# B&R Automation Studio project BaseProject
Automation Studio 4.9.2.46; technology packages: mapp 5.15.0, mappCockpit 5.15.0, mappMotion 5.15.1, mappView 5.15.1

## Configuration BuildConfig

CPU PC_any, AutomationRuntime C4.90, Build 6.3.0, Safety 0.0, Vc 

### Task classes (Cpu.sw)
```
Cyclic#8 (cycle 9600 us):
  TrakDiag <- Source.Diagnostic.TrakDiag.prg
DataObjects: McAcpSys
Binaries: McAcpDrv, udbdef, McAcpSim, mvLoader, arflatprv, McProfGen, TCLang, TCData, FWRules, mCoWebSc, arcoal, arsvcreg, McMechSys, OpcUaSrv, sysconf, Settings, FileCfg, asfw, MainAlrCfg, MachCfg, Role, ashwac, TraceConfi, iomap, AlarmHist, SectorCfg, arconfig, AsmCfg, TC, ashwd, User, ShuttleCfg, AsmFeatCfg, CoreCfg, LoggerCFG, Main, AuditCfg, Config, em2_sm2, em2_sm1, Trak
Libraries: CoTrace, AsZip, FileIO, runtime, McBase, MpAlarmX, MpBase, astime, MpFile, MpRecipe, sys_lib, McAxis, McAcpTrak, MpAxis, McAcpAx, TrBase, MpPackML, MpCom, MpServer, MpRobotics, McAxGroup, McPathGen, McProgInt, snprintf, brdkSTR, TrkPaper, ArEventLog, AsHttp, AsIODiag, AsBrStr, standard, MpAudit, McAcpPar, AdvIecChk, asstring, TrkDiag, powerlnk, asieccon, asepl, asusb, dataobj, arssl, aruser, asarprof, asmem, brsystem, asarlog, asio
```

### Hardware
```
5PC910.SX02-00 : 5PC910.SX02-00 v2.0.1.0
  Connector IF1:
    AssignedOperatingSystem = ARemb
  Connector IF3:
    AssignedOperatingSystem = ARemb
    ActivateDevice = 1
    HostName = atldemo2019
    Mode = DHCP Server
  Connector IF4:
    AssignedOperatingSystem = ARemb
    ActivateDevice = 1
    HostName = atldemo2019
    Mode = Manual
    InternetAddress = 10.1.13.45
    SubnetMask = 255.255.255.0
  Connector IF5:
    AssignedOperatingSystem = ARemb
  Connector IF6:
    AssignedOperatingSystem = ARemb
  Connector IF7:
    AssignedOperatingSystem = ARemb
  Connector IF8:
    AssignedOperatingSystem = ARemb
  Connector IF9:
    AssignedOperatingSystem = ARemb
PC : 5PC900.TS17-00 v2.1.0.0  [SY -> 5PC910.SX02-00.SY1]
  ConfigurationID = BaseProject_TestConfig
  ConfigVersion = 1.2.0
  UserPartitionSize = 1024
  Simulation = 1
  VolatileGlobalPvSize = 2000000
  SystemTick = 400
  IdleTaskClass = 3
  TaskClassIdleTime = 2400
  XLinkUseDefault = 0
  XLinkDuration = 800
  Cyclic1Duration = 800
  Cyclic1Tolerance = 0
  Cyclic1Stack = 256000
  Cyclic1Output = 1
  Cyclic2Duration = 16000
  Cyclic2Tolerance = 32000
  Cyclic2Stack = 32000
  Cyclic3Duration = 49600
  Cyclic3Tolerance = 49600
  Cyclic8Duration = 9600
  FileDevice1
  FileDeviceName1 = SvgData
  FileDevicePath1 =  ../../../../Logical/Scene/
  FileDevice2
  FileDeviceName2 = User
  FileDevicePath2 = F:\
  FileDevice3
  FileDeviceName3 = Config
  FileDevicePath3 = F:\Config\
  FileDevice4
  FileDeviceName4 = SegTraceSim
  FileDevicePath4 = ../../../../Logical/UserData/SegTrace
  FileDevice5
  FileDeviceName5 = SegTrace
  FileDevicePath5 = F:/SegTrace
  FtpUser1
  FtpUsername1 = FTP
  FtpUserPassword1 = T9zhCndb3U+RGv/CzHF4XnaM0UkBa3EbnmIr44HqX4c=  // ftpaccess
  FtpUserSalt1 = Ims2GQYk
  FTPAccessRight1 = 0
  ActivateOpcUa = 1
  OpcUaInformationModels_PV_Version = 1
```

### LoggerCFG.mappmotioncfg - PC/mappMotion/LoggerCFG.mappmotioncfg
```
Element MappMotionConfiguration (Type=mappmotioncfg)
  Logger:
    SelectiveLogging = Used
      AdministrativeCommands = Suppressed
      MovementCommands = Suppressed
      InformationalCommands = Suppressed
```

### AsmCfg.assembly - PC/mappMotion/TrakConfig/AsmCfg.assembly
```
Element gSampleTrak (Type=assembly)
  Tracks:
    TrackSeparation = 0.030
    Track[1]:
      Segments:
        SegmentRef[1] = ::gSeg_A_1
        SegmentRef[2] = ::gSeg_A_2
        SegmentRef[3] = ::gSeg_A_3
        SegmentRef[4] = ::gSeg_A_4
        SegmentRef[5] = ::gSeg_A_5
        SegmentRef[6] = ::gSeg_A_6
        SegmentRef[7] = ::gSeg_A_7
        SegmentRef[8] = ::gSeg_A_8
        SegmentRef[9] = ::gSeg_A_9
        SegmentRef[10] = ::gSeg_A_10
        SegmentRef[11] = ::gSeg_A_11
        SegmentRef[12] = ::gSeg_A_12
      Position = Absolute
        SegmentRef = ::gSeg_A_1
        SegmentCountDirection = RightToLeft
        Translation:
          X = 0.0
          Y = 0.0
          Z = 0.0
        Orientation:
          Angle1 = 0.0
          Angle2 = 0.0
          Angle3 = 0.0
    Track[2]:
      Segments:
        SegmentRef[1] = ::gSeg_B_1
        SegmentRef[2] = ::gSeg_B_2
        SegmentRef[3] = ::gSeg_B_3
        SegmentRef[4] = ::gSeg_B_4
        SegmentRef[5] = ::gSeg_B_5
        SegmentRef[6] = ::gSeg_B_6
        SegmentRef[7] = ::gSeg_B_7
        SegmentRef[8] = ::gSeg_B_8
        SegmentRef[9] = ::gSeg_B_9
        SegmentRef[10] = ::gSeg_B_10
        SegmentRef[11] = ::gSeg_B_11
      Position = RelativeToOne
        TrackSegmentPosition:
          SegmentRef = ::gSeg_B_1
        Base:
          SegmentRef = ::gSeg_A_7
  CommonSegmentSettings:
    SegmentSimulationOnPLC = Off
    ElongationCompensation = Inactive
    StopReaction = InductionHalt
    SpeedFilter = Lowpass
      FilterTime = 0.0008
    ControllerParameters:
      DefaultParameter:
        Controller:
          Position:
            ProportionalGain = 150
          Speed:
            ProportionalGain = 80
            IntegrationTime = 0.0
          FeedForward:
            TotalMass = 0.7
            ForcePositive = 1.5
            ForceNegative = 1.5
            SpeedForceFactor = 1.4
            ForceLoad = 0.0
        MovementErrorLimits:
          PositionError = 20
          VelocityError = 2000
      AdditionalParameterSets = NotUsed
    ScopeOfErrorReaction = Assembly
    ShuttleIdentificationTime = 0
  Shuttles:
    MaxShuttleCount = 20
    DistanceReserve:
      Collision = 0.002
      ErrorStop = 0.006
    ShuttleStereotypes:
      ShuttleStRef[1] = gSampleShuttle
    MagnetPlateConfigurations:
      ShuttleType[1] = 8F1SA.100.xxxxxx-x
    CollisionAvoidance:
      Strategy = Constant
      MaximumModelDimensions:
        Length:
          ExtentToFront = 0.025
          ExtentToBack = 0.025
        Width:
          Width = 0.040
  AssemblyFeatures:
    AssemblyFeatureRef[1] = SampleTrak_AutoAttach
    AssemblyFeatureRef[2] = SampleTrak_LocalLimits
    AssemblyFeatureRef[3] = SampleTrak_SimShuttle
  Visualization:
    MonitoringPv = ::gSampleTrakMon
    ProcessingTaskClass = 1
```

### AsmFeatCfg.assemblyfeature - PC/mappMotion/TrakConfig/AsmFeatCfg.assemblyfeature
```
Element SampleTrak_AutoAttach (Type=assemblyfeature)
  Type = ShtSectorAutoAttach
    Priority[1]:
      SectorRef = gSampleTrak_SectorTrakA
      Orientation = KeepSegment
Element SampleTrak_LocalLimits (Type=assemblyfeature)
  Type = LocalLimits
    LocalLimit[1]:
      Location:
        SectorRef = gSampleTrak_SectorTrakA
      MotionLimits:
        Velocity = Basic
          Velocity = 3
        Acceleration = Basic
          Acceleration = 10
Element SampleTrak_SimShuttle (Type=assemblyfeature)
  Type = InitShuttleSim
    InitShuttleSim[1]:
      SectorRef = gSampleTrak_SectorTrakA
      Orientation = Positive
      ShuttleDefinition = ShuttleSetDefinition
        StartPosition = 0.0
        NumberOfShuttles = 10
        DistnaceBetweenShuttles = 100
```

### SectorCfg.sector - PC/mappMotion/TrakConfig/SectorCfg.sector
```
Element gSampleTrak_SectorTrakB (Type=sector)
  Type = Composed
    StartSegment:
      SegmentRef = ::gSeg_B_1
    IntermediateSegments:
      SegmentRef[1] = ::gSeg_B_2
      SegmentRef[2] = ::gSeg_B_3
      SegmentRef[3] = ::gSeg_B_4
      SegmentRef[4] = ::gSeg_B_5
      SegmentRef[5] = ::gSeg_B_6
      SegmentRef[6] = ::gSeg_B_7
      SegmentRef[7] = ::gSeg_B_8
      SegmentRef[8] = ::gSeg_B_9
      SegmentRef[9] = ::gSeg_B_10
    EndSegment:
      SegmentRef = ::gSeg_B_11
      PositionRelativeTo = FromEnd
Element gSampleTrak_SectorTrakAll (Type=sector)
  Type = Composed
    StartSegment:
      SegmentRef = ::gSeg_B_4
    IntermediateSegments:
      SegmentRef[1] = ::gSeg_B_5
      SegmentRef[2] = ::gSeg_B_6
      SegmentRef[3] = ::gSeg_B_7
      SegmentRef[4] = ::gSeg_B_8
      SegmentRef[5] = ::gSeg_B_9
      SegmentRef[6] = ::gSeg_B_10
      SegmentRef[7] = ::gSeg_B_11
      SegmentRef[8] = ::gSeg_A_7
      SegmentRef[9] = ::gSeg_A_6
      SegmentRef[10] = ::gSeg_A_5
      SegmentRef[11] = ::gSeg_A_4
      SegmentRef[12] = ::gSeg_A_3
      SegmentRef[13] = ::gSeg_A_2
      SegmentRef[14] = ::gSeg_A_1
      SegmentRef[15] = ::gSeg_A_12
      SegmentRef[16] = ::gSeg_A_11
      SegmentRef[17] = ::gSeg_A_10
      SegmentRef[18] = ::gSeg_A_9
      SegmentRef[19] = ::gSeg_A_8
      SegmentRef[20] = ::gSeg_A_7
      SegmentRef[21] = ::gSeg_B_1
      SegmentRef[22] = ::gSeg_B_2
      SegmentRef[23] = ::gSeg_B_3
    EndSegment:
      SegmentRef = ::gSeg_B_4
Element gSampleTrak_SectorTrakA (Type=sector)
  Type = Composed
    StartSegment:
      SegmentRef = ::gSeg_A_1
    IntermediateSegments:
      SegmentRef[1] = ::gSeg_A_2
      SegmentRef[2] = ::gSeg_A_3
      SegmentRef[3] = ::gSeg_A_4
      SegmentRef[4] = ::gSeg_A_5
      SegmentRef[5] = ::gSeg_A_6
      SegmentRef[6] = ::gSeg_A_7
      SegmentRef[7] = ::gSeg_A_8
      SegmentRef[8] = ::gSeg_A_9
      SegmentRef[9] = ::gSeg_A_10
      SegmentRef[10] = ::gSeg_A_11
    EndSegment:
      SegmentRef = ::gSeg_A_12
      PositionRelativeTo = FromEnd
```

### AlarmHist.mpalarmxhistory - PC/mappServices/Alarm/AlarmHist.mpalarmxhistory
```
Element gAlarmXHistory (Type=mpalarmxhistory)
```

### FileCfg.mpfilemanager - PC/mappServices/MachineConfig/FileCfg.mpfilemanager
```
Element FileManagement (Type=mpfilemanager)
  FileManager:
    USB = 1
```

### CoreCFG.mppackmlcore - PC/mappServices/Operation/CoreCFG.mppackmlcore
```
Element gPackMLCore (Type=mppackmlcore)
  Operation:
    Mode = 0
  Modes:
    Mode[1]:
      ModeID = 1
      Name = Production
  Unit:
    StartupActiveMode = 1
  UnitModes:
    Mode[1]:
      ModeID = 1
  Alarms = MpAlarmX
```

## Configuration TestConfig

CPU PC_any, AutomationRuntime C4.90, Build 6.3.0, Safety 0.0, Vc 

### Task classes (Cpu.sw)
```
Cyclic#1 (cycle 800 us, tolerance 0 us):
  GlobalSetu <- Source.GlobalSetup.prg
  TSM <- Source.TSM.prg
Cyclic#2 (cycle 1600 us, tolerance 0 us):
  TSMMain <- Source.TSMMain.prg
Cyclic#3:
  TSMAlarm <- Source.TSMAlarm.prg
DataObjects: McAcpSys
Binaries: McAcpDrv, udbdef, McAcpSim, mvLoader, arflatprv, McProfGen, TCLang, TCData, FWRules, mCoWebSc, arcoal, arsvcreg, McMechSys, sysconf, Settings, FileCfg, asfw, MainAlrCfg, MachCfg, Role, ashwac, TraceConfi, iomap, AlarmHist, SectorCfg, arconfig, AsmCfg, TC, ashwd, User, ShuttleCfg, AsmFeatCfg, CoreCfg, LoggerCFG, Main, AuditCfg, Config, em2_sm2, em2_sm1, Trak
Libraries: CoTrace, AsZip, FileIO, runtime, McBase, MpAlarmX, MpBase, astime, MpFile, MpRecipe, sys_lib, McAxis, McAcpTrak, MpAxis, McAcpAx, TrBase, MpPackML, MpCom, MpServer, MpRobotics, McAxGroup, McPathGen, McProgInt, snprintf, brdkSTR, TrkPaper, ArEventLog, AsHttp, AsIODiag, AsBrStr, standard, MpAudit, McAcpPar, AdvIecChk, asstring, TrkDiag, powerlnk, asieccon, asepl, asusb, dataobj, arssl, aruser, asarprof, asmem, brsystem, asarlog
```

### Task classes (Diag.sw)
```
Cyclic#2 (cycle 1600 us, tolerance 0 us):
  DiagConfig <- Source.SampleTrak.Diagnostic.DiagConfig.prg
Cyclic#3:
  DiagAlarm <- Source.SampleTrak.Diagnostic.DiagAlarm.prg
Cyclic#8 (cycle 4800 us):
  TrackDiag <- Source.SampleTrak.Diagnostic.TrackDiag.prg
  Logbook <- Source.SampleTrak.Diagnostic.Logbook.prg
```

### Task classes (SubMod1.sw)
```
Cyclic#1 (cycle 800 us, tolerance 0 us):
  Process <- Source.SampleTrak.EMx.Process.prg
Binaries: EM12PML, EM12CFG, submod1, EM12ALM
```

### Task classes (TrakModule.sw)
```
Cyclic#1 (cycle 800 us, tolerance 0 us):
  ShuttleIni <- Source.SampleTrak.Assembly.SubModule1.ShuttleInit.prg
  AsmSampleT <- Source.SampleTrak.Assembly.AsmSampleTrak.prg
Binaries: trakmodule, TrakALM, TrakPML, TrakCFG
```

### Task classes (EM2.sw)
```
Cyclic#1 (cycle 800 us, tolerance 0 us):
  Config2 <- Source.SampleTrak.ReusableSource.Config.prg
Cyclic#2 (cycle 1600 us, tolerance 0 us):
  Operation2 <- Source.SampleTrak.ReusableSource.Operation.prg
  Alarm2 <- Source.SampleTrak.ReusableSource.Alarm.prg
Cyclic#3:
  Recovery2 <- Source.SampleTrak.ReusableSource.Recovery.prg
  BarrierCt2 <- Source.SampleTrak.ReusableSource.BarrierCtrl.prg
Binaries: em2
```

### Task classes (EM3.sw)
```
Cyclic#1 (cycle 800 us, tolerance 0 us):
  Config3 <- Source.SampleTrak.ReusableSource.Config.prg
Cyclic#2 (cycle 1600 us, tolerance 0 us):
  Operation3 <- Source.SampleTrak.ReusableSource.Operation.prg
  Alarm3 <- Source.SampleTrak.ReusableSource.Alarm.prg
Cyclic#3:
  Recovery3 <- Source.SampleTrak.ReusableSource.Recovery.prg
  BarrierCt3 <- Source.SampleTrak.ReusableSource.BarrierCtrl.prg
Binaries: em3
```

### Task classes (EMx.sw)
```
Cyclic#1 (cycle 800 us, tolerance 0 us):
  ConfigEMx <- Source.SampleTrak.EMx.Config.prg
  ProcessEMx <- Source.SampleTrak.EMx.Process.prg
Cyclic#2 (cycle 1600 us, tolerance 0 us):
  AlarmEMx <- Source.SampleTrak.EMx.Alarm.prg
Binaries: EM12PML, EM12CFG, submod1, EM12ALM
```

### Task classes (EM2.sw)
```
Cyclic#2 (cycle 1600 us, tolerance 0 us):
  Operation2 <- Source.SampleTrak.ReusableSource.Operation.prg
Binaries: em2
```

### Task classes (EM3.sw)
```
Cyclic#2 (cycle 1600 us, tolerance 0 us):
  Operation3 <- Source.SampleTrak.ReusableSource.Operation.prg
Binaries: em3
```

### Task classes (TrackMod.sw)
```
Cyclic#1 (cycle 800 us, tolerance 0 us):
  ShuttleIni <- Source.SampleTrak.Assembly.SubModule1.ShuttleInit.prg
  AsmSampleT <- Source.SampleTrak.Assembly.AsmSampleTrak.prg
  AsmConfig <- Source.SampleTrak.Assembly.AsmConfig.prg
Cyclic#3:
  AsmAlarm <- Source.SampleTrak.Assembly.AsmAlarm.prg
Binaries: trakmodule, TrakALM, TrakPML, TrakCFG
```

### Task classes (TrakMod.sw)
```
Cyclic#1 (cycle 800 us, tolerance 0 us):
  ShuttleIni <- Source.Assembly.SubModule1.ShuttleInit.prg
  AsmSampleT <- Source.Assembly.AsmSampleTrak.prg
  AsmConfig <- Source.Assembly.AsmConfig.prg
Cyclic#3:
  AsmAlarm <- Source.Assembly.AsmAlarm.prg
Binaries: trakmodule, TrakALM, TrakPML, TrakCFG
```

### Task classes (TrakModule.sw)
```
Cyclic#1 (cycle 800 us, tolerance 0 us):
  ShuttleIni <- Source.SampleTrak.Assembly.SubModule1.ShuttleInit.prg
  AsmSampleT <- Source.SampleTrak.Assembly.AsmSampleTrak.prg
Cyclic#3:
  Alarm <- Source.SampleTrak.Assembly.Alarm.prg
Binaries: trakmodule, TrakALM, TrakPML, TrakCFG
```

### Hardware
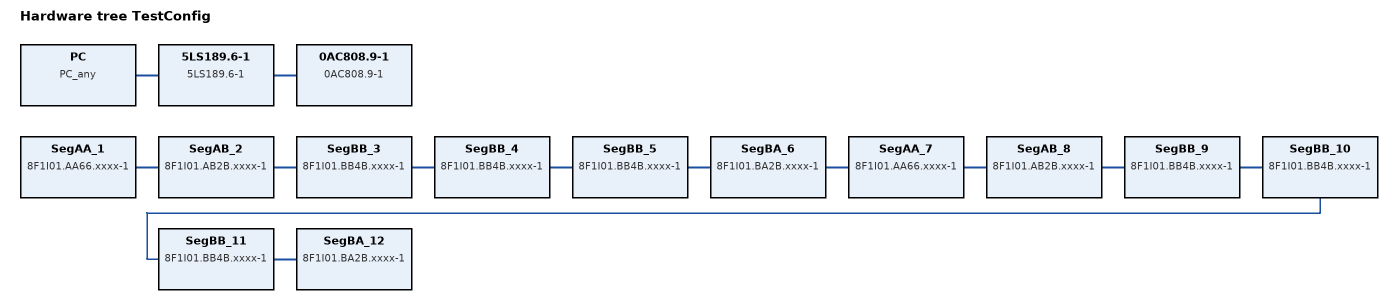
```
0AC808.9-1 : 0AC808.9-1 v1.0.0.0  [ETH1 -> 5LS189.6-1.IF2 [Cable Type=PowerlinkCable, Length=10, Version=1.0.0.3]; ETH5 -> SegAA_1.PLK3 [Cable Type=PowerlinkCable, Length=10, Version=1.0.0.3]]
5LS189.6-1 : 5LS189.6-1 v1.4.1.0  [SL -> PC.SL1]
  Connector IF2:
    CycleTime = 800
PC : PC_any v1.1.1.0 (OrderNumber=PC)
  ConfigurationID = BaseProject_TestConfig
  ConfigVersion = 1.0.0
  VolatileGlobalPvSize = 2000000
  SystemTick = 800
  Cyclic1Duration = 800
  Cyclic1Tolerance = 0
  Cyclic1Stack = 32000
  Cyclic2Duration = 1600
  Cyclic2Tolerance = 0
  Cyclic2Stack = 32000
  Cyclic8Duration = 4800
  FileDevice1
  FileDeviceName1 = SvgData
  FileDevicePath1 =  ../../../../Logical/Scene/
  FileDevice2
  FileDeviceName2 = User
  FileDevicePath2 = F:\
  FileDevice3
  FileDeviceName3 = Config
  FileDevicePath3 = F:\Config\
  FileDevice4
  FileDeviceName4 = SegTraceSim
  FileDevicePath4 = ../../../../Logical/UserData/SegTrace
  FileDevice5
  FileDeviceName5 = SegTrace
  FileDevicePath5 = F:/SegTrace
  FtpUser1
  FtpUsername1 = FTP
  FtpUserPassword1 = T9zhCndb3U+RGv/CzHF4XnaM0UkBa3EbnmIr44HqX4c=  // ftpaccess
  FtpUserSalt1 = Ims2GQYk
  FTPAccessRight1 = 0
  ActivateOpcUa = 1
  OpcUaInformationModels_PV_Version = 2
SegAA_1 : 8F1I01.AA66.xxxx-1 v1.0.0.2  [PLK2 -> SegAB_2.PLK1 (NodeNumber=1) [Cable Type=PowerlinkCable, Length=10, Version=1.0.0.3]; PLK3 -> 0AC808.9-1.ETH5 (NodeNumber=1) [Cable Type=PowerlinkCable, Length=10, Version=1.0.0.3]]
  DriveConfiguration:
    McTypeID = LLMConfig
  DriveConfiguration/Segment:
    Shape = STRAIGHT660
    SegmentReference = gSeg_A_1
    StopReaction = UseAssemblySetting
    SpeedFilter = UseAssemblySetting
SegAA_7 : 8F1I01.AA66.xxxx-1 v1.0.0.2  [PLK1 -> SegBA_6.PLK2 [Cable Type=PowerlinkCable, Length=10, Version=1.0.0.3]; PLK2 -> SegAB_8.PLK1 [Cable Type=PowerlinkCable, Length=10, Version=1.0.0.3]]
  DriveConfiguration:
    McTypeID = LLMConfig
  DriveConfiguration/Segment:
    Shape = STRAIGHT660
    SegmentReference = gSeg_A_7
    StopReaction = UseAssemblySetting
    SpeedFilter = UseAssemblySetting
SegAB_2 : 8F1I01.AB2B.xxxx-1 v1.0.0.2  [PLK1 -> SegAA_1.PLK2 [Cable Type=PowerlinkCable, Length=10, Version=1.0.0.3]; PLK2 -> SegBB_3.PLK1 [Cable Type=PowerlinkCable, Length=10, Version=1.0.0.3]]
  DriveConfiguration:
    McTypeID = LLMConfig
  DriveConfiguration/Segment:
    Shape = STRAIGHT105_TO_CIRCULAR
    SegmentReference = gSeg_A_2
    StopReaction = UseAssemblySetting
    SpeedFilter = UseAssemblySetting
SegAB_8 : 8F1I01.AB2B.xxxx-1 v1.0.0.2  [PLK1 -> SegAA_7.PLK2 [Cable Type=PowerlinkCable, Length=10, Version=1.0.0.3]; PLK2 -> SegBB_9.PLK1 [Cable Type=PowerlinkCable, Length=10, Version=1.0.0.3]]
  DriveConfiguration:
    McTypeID = LLMConfig
  DriveConfiguration/Segment:
    Shape = STRAIGHT105_TO_CIRCULAR
    SegmentReference = gSeg_A_8
    StopReaction = UseAssemblySetting
    SpeedFilter = UseAssemblySetting
SegBA_12 : 8F1I01.BA2B.xxxx-1 v1.0.0.2  [PLK1 -> SegBB_11.PLK2 [Cable Type=PowerlinkCable, Length=10, Version=1.0.0.3]]
  DriveConfiguration:
    McTypeID = LLMConfig
  DriveConfiguration/Segment:
    Shape = CIRCULAR_TO_STRAIGHT105
    SegmentReference = gSeg_A_12
    StopReaction = UseAssemblySetting
    SpeedFilter = UseAssemblySetting
SegBA_6 : 8F1I01.BA2B.xxxx-1 v1.0.0.2  [PLK1 -> SegBB_5.PLK2 [Cable Type=PowerlinkCable, Length=10, Version=1.0.0.3]; PLK2 -> SegAA_7.PLK1 [Cable Type=PowerlinkCable, Length=10, Version=1.0.0.3]]
  DriveConfiguration:
    McTypeID = LLMConfig
  DriveConfiguration/Segment:
    Shape = CIRCULAR_TO_STRAIGHT105
    SegmentReference = gSeg_A_6
    StopReaction = UseAssemblySetting
    SpeedFilter = UseAssemblySetting
SegBB_10 : 8F1I01.BB4B.xxxx-1 v1.0.0.2  [PLK1 -> SegBB_9.PLK2 [Cable Type=PowerlinkCable, Length=10, Version=1.0.0.3]; PLK2 -> SegBB_11.PLK1 [Cable Type=PowerlinkCable, Length=10, Version=1.0.0.3]]
  DriveConfiguration:
    McTypeID = LLMConfig
  DriveConfiguration/Segment:
    Shape = CIRCULAR
    SegmentReference = gSeg_A_10
    StopReaction = UseAssemblySetting
    SpeedFilter = UseAssemblySetting
SegBB_11 : 8F1I01.BB4B.xxxx-1 v1.0.0.2  [PLK1 -> SegBB_10.PLK2 (NodeNumber=11) [Cable Type=PowerlinkCable, Length=10, Version=1.0.0.3]; PLK2 -> SegBA_12.PLK1 (NodeNumber=11) [Cable Type=PowerlinkCable, Length=10, Version=1.0.0.3]]
  DriveConfiguration:
    McTypeID = LLMConfig
  DriveConfiguration/Segment:
    Shape = CIRCULAR
    SegmentReference = gSeg_A_11
    StopReaction = UseAssemblySetting
    SpeedFilter = UseAssemblySetting
SegBB_3 : 8F1I01.BB4B.xxxx-1 v1.0.0.2  [PLK1 -> SegAB_2.PLK2 [Cable Type=PowerlinkCable, Length=10, Version=1.0.0.3]; PLK2 -> SegBB_4.PLK1 [Cable Type=PowerlinkCable, Length=10, Version=1.0.0.3]]
  DriveConfiguration:
    McTypeID = LLMConfig
  DriveConfiguration/Segment:
    Shape = CIRCULAR
    SegmentReference = gSeg_A_3
    StopReaction = UseAssemblySetting
    SpeedFilter = UseAssemblySetting
SegBB_4 : 8F1I01.BB4B.xxxx-1 v1.0.0.2  [PLK1 -> SegBB_3.PLK2 [Cable Type=PowerlinkCable, Length=10, Version=1.0.0.3]; PLK2 -> SegBB_5.PLK1 [Cable Type=PowerlinkCable, Length=10, Version=1.0.0.3]]
  DriveConfiguration:
    McTypeID = LLMConfig
  DriveConfiguration/Segment:
    Shape = CIRCULAR
    SegmentReference = gSeg_A_4
    StopReaction = UseAssemblySetting
    SpeedFilter = UseAssemblySetting
SegBB_5 : 8F1I01.BB4B.xxxx-1 v1.0.0.2  [PLK1 -> SegBB_4.PLK2 [Cable Type=PowerlinkCable, Length=10, Version=1.0.0.3]; PLK2 -> SegBA_6.PLK1 [Cable Type=PowerlinkCable, Length=10, Version=1.0.0.3]]
  DriveConfiguration:
    McTypeID = LLMConfig
  DriveConfiguration/Segment:
    Shape = CIRCULAR
    SegmentReference = gSeg_A_5
    StopReaction = UseAssemblySetting
    SpeedFilter = UseAssemblySetting
SegBB_9 : 8F1I01.BB4B.xxxx-1 v1.0.0.2  [PLK1 -> SegAB_8.PLK2 [Cable Type=PowerlinkCable, Length=10, Version=1.0.0.3]; PLK2 -> SegBB_10.PLK1 [Cable Type=PowerlinkCable, Length=10, Version=1.0.0.3]]
  DriveConfiguration:
    McTypeID = LLMConfig
  DriveConfiguration/Segment:
    Shape = CIRCULAR
    SegmentReference = gSeg_A_9
    StopReaction = UseAssemblySetting
    SpeedFilter = UseAssemblySetting
```

### Diag.vvm - PC/Diag/Diag.vvm
```iecst
VAR_CONFIG
	Cyclic#1.Diag::gRecipeXml_DiagModule AT %Q.Cyclic#1.Diag::DiagInterface.RecipeCore; (*Insert your comment here...*)
	Cyclic#1.Diag::gAuditTrail_DiagModule AT %Q.Cyclic#1.Diag::DiagInterface.AuditCore; (*Insert your comment here...*)
	Cyclic#1.Diag::gAlarmXCore_DiagModule AT %Q.Cyclic#1.Diag::DiagInterface.AlarmCore; (*Insert your comment here...*)
	Cyclic#1.::gSampleTrak AT %Q.Cyclic#1.Diag::DiagInterface.SampleTrak; (*Insert your comment here...*)
	Cyclic#1.::gSampleTrakMon AT %Q.Cyclic#1.Diag::DiagInterface.ShuttleMon; (*Insert your comment here...*)
	Cyclic#1.::gTrakData.Seg AT %Q.Cyclic#1.Diag::TrakDiag:TrakDiag.Seg; (*Insert your comment here...*)
	Cyclic#1.TrakMod::gTrakSystem AT %Q.Cyclic#1.Diag::DiagInterface.TrakInterface; (*Insert your comment here...*)
END_VAR
```

### DiagALM.mpalarmxcore - PC/Diag/mappServices/DiagALM.mpalarmxcore
```
Element gAlarmXCore_DiagModule (Type=mpalarmxcore)
  mapp.AlarmX.Core:
    Mapping:
      [0]:
        Alarm = Inf*
        [0] = Aggregate
          Name = DiagModuleInfo
        [1]
        [2]
      [1]:
        Alarm = Warn*
        [0] = Aggregate
          Name = DiagModuleWarning
        [1]
        [2]
      [2]:
        Alarm = Alrm*
        [0] = Aggregate
          Name = DiagModuleAlarm
        [1]
        [2]
      [3]:
        Alarm = EventID*
        [0] = Aggregate
          Name = InternalTrakError
    Default:
      [0] = Remain
  mapp.AlarmX.Core.Configuration:
    [0]:
      Name = Inf_ModuleTest
      Message = {$Diag/LocalDiagModuleInfo}
      Severity = 0
      Behavior = DiscreteValueMonitoring
        Monitoring:
          MonitoredPV = Diag::DiagAlarm:TriggerTestInformation
          TriggerValues:
            [0] = TRUE
    [1]:
      Name = Warn_ModuleTest
      Message = {$Diag/LocalDiagModuleWarning}
      Code = 100
      Severity = 50
      Behavior = DiscreteValueMonitoring
        Monitoring:
          MonitoredPV = Diag::DiagAlarm:TriggerTestWarning
          TriggerValues:
            [0] = TRUE
    [2]:
      Name = Alrm_ModuleTest
      Message = {$Diag/LocalDiagModuleAlarm}
      Code = 1000
      Severity = 100
      Behavior = DiscreteValueMonitoring
        Monitoring:
          MonitoredPV = Diag::DiagAlarm:TriggerTestAlarm
          TriggerValues:
            [0] = TRUE
    [3]:
      Name = DiagModuleInfo
      Message = {$Diag/Module.Info}
      AdditionalInformation1 = diagAlarmContent
    [4]:
      Name = DiagModuleWarning
      Message = {$Diag/Module.Warning}
      Code = 100
      AdditionalInformation1 = diagAlarmContent
    [5]:
      Name = DiagModuleAlarm
      Message = {$Diag/Module.Alarm}
      Code = 1000
      AdditionalInformation1 = diagAlarmContent
    [6]:
      Name = InternalTrakError
      Message = {$Diag/Module.Error}
      Code = 1000
      AdditionalInformation1 = diagAlarmContent
    [7]:
      Name = EventIDCode.1
      Message = {$IAT/TrakError/Code.1} Count: {&Cnt.1} | {$IAT/TrakError/CheckLogBook}
      Behavior = UserDefined
        AutoReset = TRUE
        DataUpdate:
          Activation:
            TimeStamp = TRUE
            Snippets = TRUE
        Recording:
          ActiveToInactive = FALSE
          AcknowledgedToUnacknowledged = FALSE
    [8]:
      Name = EventIDCode.2
      Message = {$IAT/TrakError/Code.2} Count: {&Cnt.2} | {$IAT/TrakError/CheckLogBook}
      Behavior = UserDefined
        AutoReset = TRUE
        DataUpdate:
          Activation:
            TimeStamp = TRUE
            Snippets = TRUE
        Recording:
          ActiveToInactive = FALSE
          AcknowledgedToUnacknowledged = FALSE
    [9]:
      Name = EventIDCode.7
      Message = {$IAT/TrakError/Code.7} Count: {&Cnt.7} | {$IAT/TrakError/CheckLogBook}
      Behavior = UserDefined
        AutoReset = TRUE
        DataUpdate:
          Activation:
            TimeStamp = TRUE
            Snippets = TRUE
        Recording:
          ActiveToInactive = FALSE
          AcknowledgedToUnacknowledged = FALSE
    [10]:
      Name = EventIDCode.2048
      Message = {$IAT/TrakError/Code.2048} Count: {&Cnt.2048} | {$IAT/TrakError/CheckLogBook}
      Behavior = UserDefined
        AutoReset = TRUE
        DataUpdate:
          Activation:
            TimeStamp = TRUE
            Snippets = TRUE
        Recording:
          ActiveToInactive = FALSE
          AcknowledgedToUnacknowledged = FALSE
    [11]:
      Name = EventIDCode.2049
      Message = {$IAT/TrakError/Code.2049} Count: {&Cnt.2049} | {$IAT/TrakError/CheckLogBook}
      Behavior = UserDefined
        AutoReset = TRUE
        DataUpdate:
          Activation:
            TimeStamp = TRUE
            Snippets = TRUE
        Recording:
          ActiveToInactive = FALSE
          AcknowledgedToUnacknowledged = FALSE
    [12]:
      Name = EventIDCode.2050
      Message = {$IAT/TrakError/Code.2050} Count: {&Cnt.2050} | {$IAT/TrakError/CheckLogBook}
      Behavior = UserDefined
        AutoReset = TRUE
        DataUpdate:
          Activation:
            TimeStamp = TRUE
            Snippets = TRUE
        Recording:
          ActiveToInactive = FALSE
          AcknowledgedToUnacknowledged = FALSE
    [13]:
      Name = EventIDCode.2051
      Message = {$IAT/TrakError/Code.2051} Count: {&Cnt.2051} | {$IAT/TrakError/CheckLogBook}
      Behavior = UserDefined
        AutoReset = TRUE
        DataUpdate:
          Activation:
            TimeStamp = TRUE
            Snippets = TRUE
        Recording:
          ActiveToInactive = FALSE
          AcknowledgedToUnacknowledged = FALSE
    [14]:
      Name = EventIDCode.2052
      Message = {$IAT/TrakError/Code.2052} Count: {&Cnt.2052} | {$IAT/TrakError/CheckLogBook}
      Behavior = UserDefined
        AutoReset = TRUE
        DataUpdate:
          Activation:
            TimeStamp = TRUE
            Snippets = TRUE
        Recording:
          ActiveToInactive = FALSE
          AcknowledgedToUnacknowledged = FALSE
    [15]:
      Name = EventIDCode.2053
      Message = {$IAT/TrakError/Code.2053} Count: {&Cnt.2053} | {$IAT/TrakError/CheckLogBook}
      Behavior = UserDefined
        AutoReset = TRUE
        DataUpdate:
          Activation:
            TimeStamp = TRUE
            Snippets = TRUE
        Recording:
          ActiveToInactive = FALSE
          AcknowledgedToUnacknowledged = FALSE
    [16]:
      Name = EventIDCode.2054
      Message = {$IAT/TrakError/Code.2054} Count: {&Cnt.2054} | {$IAT/TrakError/CheckLogBook}
      Behavior = UserDefined
        AutoReset = TRUE
        DataUpdate:
          Activation:
            TimeStamp = TRUE
            Snippets = TRUE
        Recording:
          ActiveToInactive = FALSE
          AcknowledgedToUnacknowledged = FALSE
    [17]:
      Name = EventIDCode.2055
      Message = {$IAT/TrakError/Code.2055} Count: {&Cnt.2055} | {$IAT/TrakError/CheckLogBook}
      Behavior = UserDefined
        AutoReset = TRUE
        DataUpdate:
          Activation:
            TimeStamp = TRUE
            Snippets = TRUE
        Recording:
          ActiveToInactive = FALSE
          AcknowledgedToUnacknowledged = FALSE
    [18]:
      Name = EventIDCode.2056
      Message = {$IAT/TrakError/Code.2056} Count: {&Cnt.2056} | {$IAT/TrakError/CheckLogBook}
      Behavior = UserDefined
        AutoReset = TRUE
        DataUpdate:
          Activation:
            TimeStamp = TRUE
            Snippets = TRUE
        Recording:
          ActiveToInactive = FALSE
          AcknowledgedToUnacknowledged = FALSE
    [19]:
      Name = EventIDCode.2057
      Message = {$IAT/TrakError/Code.2057} Count: {&Cnt.2057} | {$IAT/TrakError/CheckLogBook}
      Behavior = UserDefined
        AutoReset = TRUE
        DataUpdate:
          Activation:
            TimeStamp = TRUE
            Snippets = TRUE
        Recording:
          ActiveToInactive = FALSE
          AcknowledgedToUnacknowledged = FALSE
    [20]:
      Name = EventIDCode.2058
      Message = {$IAT/TrakError/Code.2058} Count: {&Cnt.2058} | {$IAT/TrakError/CheckLogBook}
      Behavior = UserDefined
        AutoReset = TRUE
        DataUpdate:
          Activation:
            TimeStamp = TRUE
            Snippets = TRUE
        Recording:
          ActiveToInactive = FALSE
          AcknowledgedToUnacknowledged = FALSE
    [21]:
      Name = EventIDCode.2060
      Message = {$IAT/TrakError/Code.2060} Count: {&Cnt.2060} | {$IAT/TrakError/CheckLogBook}
      Behavior = UserDefined
        AutoReset = TRUE
        DataUpdate:
          Activation:
            TimeStamp = TRUE
            Snippets = TRUE
        Recording:
          ActiveToInactive = FALSE
          AcknowledgedToUnacknowledged = FALSE
    [22]:
      Name = EventIDCode.2061
      Message = {$IAT/TrakError/Code.2061} Count: {&Cnt.2061} | {$IAT/TrakError/CheckLogBook}
      Behavior = UserDefined
        AutoReset = TRUE
        DataUpdate:
          Activation:
            TimeStamp = TRUE
            Snippets = TRUE
        Recording:
          ActiveToInactive = FALSE
          AcknowledgedToUnacknowledged = FALSE
    [23]:
      Name = EventIDCode.2063
      Message = {$IAT/TrakError/Code.2063} Count: {&Cnt.2063} | {$IAT/TrakError/CheckLogBook}
      Behavior = UserDefined
        AutoReset = TRUE
        DataUpdate:
          Activation:
            TimeStamp = TRUE
            Snippets = TRUE
        Recording:
          ActiveToInactive = FALSE
          AcknowledgedToUnacknowledged = FALSE
    [24]:
      Name = EventIDCode.2064
      Message = {$IAT/TrakError/Code.2064} Count: {&Cnt.2064} | {$IAT/TrakError/CheckLogBook}
      Behavior = UserDefined
        AutoReset = TRUE
        DataUpdate:
          Activation:
            TimeStamp = TRUE
            Snippets = TRUE
        Recording:
          ActiveToInactive = FALSE
          AcknowledgedToUnacknowledged = FALSE
    [25]:
      Name = EventIDCode.2066
      Message = {$IAT/TrakError/Code.2066} Count: {&Cnt.2066} | {$IAT/TrakError/CheckLogBook}
      Behavior = UserDefined
        AutoReset = TRUE
        DataUpdate:
          Activation:
            TimeStamp = TRUE
            Snippets = TRUE
        Recording:
          ActiveToInactive = FALSE
          AcknowledgedToUnacknowledged = FALSE
    [26]:
      Name = EventIDCode.2067
      Message = {$IAT/TrakError/Code.2067} Count: {&Cnt.2067} | {$IAT/TrakError/CheckLogBook}
      Behavior = UserDefined
        AutoReset = TRUE
        DataUpdate:
          Activation:
            TimeStamp = TRUE
            Snippets = TRUE
        Recording:
          ActiveToInactive = FALSE
          AcknowledgedToUnacknowledged = FALSE
    [27]:
      Name = EventIDCode.2068
      Message = {$IAT/TrakError/Code.2068} Count: {&Cnt.2068} | {$IAT/TrakError/CheckLogBook}
      Behavior = UserDefined
        AutoReset = TRUE
        DataUpdate:
          Activation:
            TimeStamp = TRUE
            Snippets = TRUE
        Recording:
          ActiveToInactive = FALSE
          AcknowledgedToUnacknowledged = FALSE
    [28]:
      Name = EventIDCode.2069
      Message = {$IAT/TrakError/Code.2069} Count: {&Cnt.2069} | {$IAT/TrakError/CheckLogBook}
      Behavior = UserDefined
        AutoReset = TRUE
        DataUpdate:
          Activation:
            TimeStamp = TRUE
            Snippets = TRUE
        Recording:
          ActiveToInactive = FALSE
          AcknowledgedToUnacknowledged = FALSE
    [29]:
      Name = EventIDCode.2070
      Message = {$IAT/TrakError/Code.2070} Count: {&Cnt.2070} | {$IAT/TrakError/CheckLogBook}
      Behavior = UserDefined
        AutoReset = TRUE
        DataUpdate:
          Activation:
            TimeStamp = TRUE
            Snippets = TRUE
        Recording:
          ActiveToInactive = FALSE
          AcknowledgedToUnacknowledged = FALSE
    [30]:
      Name = EventIDCode.2071
      Message = {$IAT/TrakError/Code.2071} Count: {&Cnt.2071} | {$IAT/TrakError/CheckLogBook}
      Behavior = UserDefined
        AutoReset = TRUE
        DataUpdate:
          Activation:
            TimeStamp = TRUE
            Snippets = TRUE
        Recording:
          ActiveToInactive = FALSE
          AcknowledgedToUnacknowledged = FALSE
    [31]:
      Name = EventIDCode.2074
      Message = {$IAT/TrakError/Code.2074} Count: {&Cnt.2074} | {$IAT/TrakError/CheckLogBook}
      Behavior = UserDefined
        AutoReset = TRUE
        DataUpdate:
          Activation:
            TimeStamp = TRUE
            Snippets = TRUE
        Recording:
          ActiveToInactive = FALSE
          AcknowledgedToUnacknowledged = FALSE
    [32]:
      Name = EventIDCode.2077
      Message = {$IAT/TrakError/Code.2077} Count: {&Cnt.2077} | {$IAT/TrakError/CheckLogBook}
      Behavior = UserDefined
        AutoReset = TRUE
        DataUpdate:
          Activation:
            TimeStamp = TRUE
            Snippets = TRUE
        Recording:
          ActiveToInactive = FALSE
          AcknowledgedToUnacknowledged = FALSE
    [33]:
      Name = EventIDCode.2080
      Message = {$IAT/TrakError/Code.2080} Count: {&Cnt.2080} | {$IAT/TrakError/CheckLogBook}
      Behavior = UserDefined
        AutoReset = TRUE
        DataUpdate:
          Activation:
            TimeStamp = TRUE
            Snippets = TRUE
        Recording:
          ActiveToInactive = FALSE
          AcknowledgedToUnacknowledged = FALSE
    [34]:
      Name = EventIDCode.2082
      Message = {$IAT/TrakError/Code.2082} Count: {&Cnt.2082} | {$IAT/TrakError/CheckLogBook}
      Behavior = UserDefined
        AutoReset = TRUE
        DataUpdate:
          Activation:
            TimeStamp = TRUE
            Snippets = TRUE
        Recording:
          ActiveToInactive = FALSE
          AcknowledgedToUnacknowledged = FALSE
    [35]:
      Name = EventIDCode.2083
      Message = {$IAT/TrakError/Code.2083} Count: {&Cnt.2083} | {$IAT/TrakError/CheckLogBook}
      Behavior = UserDefined
        AutoReset = TRUE
        DataUpdate:
          Activation:
            TimeStamp = TRUE
            Snippets = TRUE
        Recording:
          ActiveToInactive = FALSE
          AcknowledgedToUnacknowledged = FALSE
    [36]:
      Name = EventIDCode.2084
      Message = {$IAT/TrakError/Code.2084} Count: {&Cnt.2084} | {$IAT/TrakError/CheckLogBook}
      Behavior = UserDefined
        AutoReset = TRUE
        DataUpdate:
          Activation:
            TimeStamp = TRUE
            Snippets = TRUE
        Recording:
          ActiveToInactive = FALSE
          AcknowledgedToUnacknowledged = FALSE
    [37]:
      Name = EventIDCode.2085
      Message = {$IAT/TrakError/Code.2085} Count: {&Cnt.2085} | {$IAT/TrakError/CheckLogBook}
      Behavior = UserDefined
        AutoReset = TRUE
        DataUpdate:
          Activation:
            TimeStamp = TRUE
            Snippets = TRUE
        Recording:
          ActiveToInactive = FALSE
          AcknowledgedToUnacknowledged = FALSE
    [38]:
      Name = EventIDCode.2090
      Message = {$IAT/TrakError/Code.2090} Count: {&Cnt.2090} | {$IAT/TrakError/CheckLogBook}
      Behavior = UserDefined
        AutoReset = TRUE
        DataUpdate:
          Activation:
            TimeStamp = TRUE
            Snippets = TRUE
        Recording:
          ActiveToInactive = FALSE
          AcknowledgedToUnacknowledged = FALSE
    [39]:
      Name = EventIDCode.2091
      Message = {$IAT/TrakError/Code.2091} Count: {&Cnt.2091} | {$IAT/TrakError/CheckLogBook}
      Behavior = UserDefined
        AutoReset = TRUE
        DataUpdate:
          Activation:
            TimeStamp = TRUE
            Snippets = TRUE
        Recording:
          ActiveToInactive = FALSE
          AcknowledgedToUnacknowledged = FALSE
    [40]:
      Name = EventIDCode.2092
      Message = {$IAT/TrakError/Code.2092} Count: {&Cnt.2092} | {$IAT/TrakError/CheckLogBook}
      Behavior = UserDefined
        AutoReset = TRUE
        DataUpdate:
          Activation:
            TimeStamp = TRUE
            Snippets = TRUE
        Recording:
          ActiveToInactive = FALSE
          AcknowledgedToUnacknowledged = FALSE
    [41]:
      Name = EventIDCode.2093
      Message = {$IAT/TrakError/Code.2093} Count: {&Cnt.2093} | {$IAT/TrakError/CheckLogBook}
      Behavior = UserDefined
        AutoReset = TRUE
        DataUpdate:
          Activation:
            TimeStamp = TRUE
            Snippets = TRUE
        Recording:
          ActiveToInactive = FALSE
          AcknowledgedToUnacknowledged = FALSE
    [42]:
      Name = EventIDCode.2094
      Message = {$IAT/TrakError/Code.2094} Count: {&Cnt.2094} | {$IAT/TrakError/CheckLogBook}
      Behavior = UserDefined
        AutoReset = TRUE
        DataUpdate:
          Activation:
            TimeStamp = TRUE
            Snippets = TRUE
        Recording:
          ActiveToInactive = FALSE
          AcknowledgedToUnacknowledged = FALSE
    [43]:
      Name = EventIDCode.2095
      Message = {$IAT/TrakError/Code.2095} Count: {&2095} | {$IAT/TrakError/CheckLogBook}
      Behavior = UserDefined
        AutoReset = TRUE
        DataUpdate:
          Activation:
            TimeStamp = TRUE
            Snippets = TRUE
        Recording:
          ActiveToInactive = FALSE
          AcknowledgedToUnacknowledged = FALSE
    [44]:
      Name = EventIDCode.2097
      Message = {$IAT/TrakError/Code.2097} Count: {&Cnt.2097} | {$IAT/TrakError/CheckLogBook}
      Behavior = UserDefined
        AutoReset = TRUE
        DataUpdate:
          Activation:
            TimeStamp = TRUE
            Snippets = TRUE
        Recording:
          ActiveToInactive = FALSE
          AcknowledgedToUnacknowledged = FALSE
    [45]:
      Name = EventIDCode.2098
      Message = {$IAT/TrakError/Code.2098} Count: {&Cnt.2098} | {$IAT/TrakError/CheckLogBook}
      Behavior = UserDefined
        AutoReset = TRUE
        DataUpdate:
          Activation:
            TimeStamp = TRUE
            Snippets = TRUE
        Recording:
          ActiveToInactive = FALSE
          AcknowledgedToUnacknowledged = FALSE
    [46]:
      Name = EventIDCode.2099
      Message = {$IAT/TrakError/Code.2099} Count: {&Cnt.2099} | {$IAT/TrakError/CheckLogBook}
      Behavior = UserDefined
        AutoReset = TRUE
        DataUpdate:
          Activation:
            TimeStamp = TRUE
            Snippets = TRUE
        Recording:
          ActiveToInactive = FALSE
          AcknowledgedToUnacknowledged = FALSE
    [47]:
      Name = EventIDCode.2100
      Message = {$IAT/TrakError/Code.2100} Count: {&Cnt.2100} | {$IAT/TrakError/CheckLogBook}
      Behavior = UserDefined
        AutoReset = TRUE
        DataUpdate:
          Activation:
            TimeStamp = TRUE
            Snippets = TRUE
        Recording:
          ActiveToInactive = FALSE
          AcknowledgedToUnacknowledged = FALSE
    [48]:
      Name = EventIDCode.2101
      Message = {$IAT/TrakError/Code.2101} Count: {&Cnt.2101} | {$IAT/TrakError/CheckLogBook}
      Behavior = UserDefined
        AutoReset = TRUE
        DataUpdate:
          Activation:
            TimeStamp = TRUE
            Snippets = TRUE
        Recording:
          ActiveToInactive = FALSE
          AcknowledgedToUnacknowledged = FALSE
    [49]:
      Name = EventIDCode.2102
      Message = {$IAT/TrakError/Code.2102} Count: {&Cnt.2102} | {$IAT/TrakError/CheckLogBook}
      Behavior = UserDefined
        AutoReset = TRUE
        DataUpdate:
          Activation:
            TimeStamp = TRUE
            Snippets = TRUE
        Recording:
          ActiveToInactive = FALSE
          AcknowledgedToUnacknowledged = FALSE
    [50]:
      Name = EventIDCode.2103
      Message = {$IAT/TrakError/Code.2103} Count: {&Cnt.2103} | {$IAT/TrakError/CheckLogBook}
      Behavior = UserDefined
        AutoReset = TRUE
        DataUpdate:
          Activation:
            TimeStamp = TRUE
            Snippets = TRUE
        Recording:
          ActiveToInactive = FALSE
          AcknowledgedToUnacknowledged = FALSE
    [51]:
      Name = EventIDCode.2104
      Message = {$IAT/TrakError/Code.2104} Count: {&Cnt.2104} | {$IAT/TrakError/CheckLogBook}
      Behavior = UserDefined
        AutoReset = TRUE
        DataUpdate:
          Activation:
            TimeStamp = TRUE
            Snippets = TRUE
        Recording:
          ActiveToInactive = FALSE
          AcknowledgedToUnacknowledged = FALSE
    [52]:
      Name = EventIDCode.2105
      Message = {$IAT/TrakError/Code.2105} Count: {&Cnt.2105} | {$IAT/TrakError/CheckLogBook}
      Behavior = UserDefined
        AutoReset = TRUE
        DataUpdate:
          Activation:
            TimeStamp = TRUE
            Snippets = TRUE
        Recording:
          ActiveToInactive = FALSE
          AcknowledgedToUnacknowledged = FALSE
    [53]:
      Name = EventIDCode.2106
      Message = {$IAT/TrakError/Code.2106} Count: {&Cnt.2106} | {$IAT/TrakError/CheckLogBook}
      Behavior = UserDefined
        AutoReset = TRUE
        DataUpdate:
          Activation:
            TimeStamp = TRUE
            Snippets = TRUE
        Recording:
          ActiveToInactive = FALSE
          AcknowledgedToUnacknowledged = FALSE
    [54]:
      Name = EventIDCode.2107
      Message = {$IAT/TrakError/Code.2107} Count: {&Cnt.2107} | {$IAT/TrakError/CheckLogBook}
      Behavior = UserDefined
        AutoReset = TRUE
        DataUpdate:
          Activation:
            TimeStamp = TRUE
            Snippets = TRUE
        Recording:
          ActiveToInactive = FALSE
          AcknowledgedToUnacknowledged = FALSE
    [55]:
      Name = EventIDCode.2108
      Message = {$IAT/TrakError/Code.2108} Count: {&Cnt.2108} | {$IAT/TrakError/CheckLogBook}
      Behavior = UserDefined
        AutoReset = TRUE
        DataUpdate:
          Activation:
            TimeStamp = TRUE
            Snippets = TRUE
        Recording:
          ActiveToInactive = FALSE
          AcknowledgedToUnacknowledged = FALSE
    [56]:
      Name = EventIDCode.2109
      Message = {$IAT/TrakError/Code.2109} Count: {&Cnt.2109} | {$IAT/TrakError/CheckLogBook}
      Behavior = UserDefined
        AutoReset = TRUE
        DataUpdate:
          Activation:
            TimeStamp = TRUE
            Snippets = TRUE
        Recording:
          ActiveToInactive = FALSE
          AcknowledgedToUnacknowledged = FALSE
    [57]:
      Name = EventIDCode.2110
      Message = {$IAT/TrakError/Code.2110} Count: {&Cnt.2110} | {$IAT/TrakError/CheckLogBook}
      Behavior = UserDefined
        AutoReset = TRUE
        DataUpdate:
          Activation:
            TimeStamp = TRUE
            Snippets = TRUE
        Recording:
          ActiveToInactive = FALSE
          AcknowledgedToUnacknowledged = FALSE
    [58]:
      Name = EventIDCode.2111
      Message = {$IAT/TrakError/Code.2111} Count: {&Cnt.2111} | {$IAT/TrakError/CheckLogBook}
      Behavior = UserDefined
        AutoReset = TRUE
        DataUpdate:
          Activation:
            TimeStamp = TRUE
            Snippets = TRUE
        Recording:
          ActiveToInactive = FALSE
          AcknowledgedToUnacknowledged = FALSE
    [59]:
      Name = EventIDCode.2112
      Message = {$IAT/TrakError/Code.2112} Count: {&Cnt.2112} | {$IAT/TrakError/CheckLogBook}
      Behavior = UserDefined
        AutoReset = TRUE
        DataUpdate:
          Activation:
            TimeStamp = TRUE
            Snippets = TRUE
        Recording:
          ActiveToInactive = FALSE
          AcknowledgedToUnacknowledged = FALSE
    [60]:
      Name = EventIDCode.4096
      Message = {$IAT/TrakError/Code.4096} Count: {&Cnt.4096} | {$IAT/TrakError/CheckLogBook}
      Behavior = UserDefined
        AutoReset = TRUE
        DataUpdate:
          Activation:
            TimeStamp = TRUE
            Snippets = TRUE
        Recording:
          ActiveToInactive = FALSE
          AcknowledgedToUnacknowledged = FALSE
    [61]:
      Name = EventIDCode.4097
      Message = {$IAT/TrakError/Code.4097} Count: {&Cnt.4097} | {$IAT/TrakError/CheckLogBook}
      Behavior = UserDefined
        AutoReset = TRUE
        DataUpdate:
          Activation:
            TimeStamp = TRUE
            Snippets = TRUE
        Recording:
          ActiveToInactive = FALSE
          AcknowledgedToUnacknowledged = FALSE
    [62]:
      Name = EventIDCode.4101
      Message = {$IAT/TrakError/Code.4101} Count: {&Cnt.4101} | {$IAT/TrakError/CheckLogBook}
      Behavior = UserDefined
        AutoReset = TRUE
        DataUpdate:
          Activation:
            TimeStamp = TRUE
            Snippets = TRUE
        Recording:
          ActiveToInactive = FALSE
          AcknowledgedToUnacknowledged = FALSE
    [63]:
      Name = EventIDCode.4102
      Message = {$IAT/TrakError/Code.4102} Count: {&Cnt.4102} | {$IAT/TrakError/CheckLogBook}
      Behavior = UserDefined
        AutoReset = TRUE
        DataUpdate:
          Activation:
            TimeStamp = TRUE
            Snippets = TRUE
        Recording:
          ActiveToInactive = FALSE
          AcknowledgedToUnacknowledged = FALSE
    [64]:
      Name = EventIDCode.6144
      Message = {$IAT/TrakError/Code.6144} Count: {&Cnt.6144} | {$IAT/TrakError/CheckLogBook}
      Behavior = UserDefined
        AutoReset = TRUE
        DataUpdate:
          Activation:
            TimeStamp = TRUE
            Snippets = TRUE
        Recording:
          ActiveToInactive = FALSE
          AcknowledgedToUnacknowledged = FALSE
    [65]:
      Name = EventIDCode.6165
      Message = {$IAT/TrakError/Code.6165} Count: {&Cnt.6165} | {$IAT/TrakError/CheckLogBook}
      Behavior = UserDefined
        AutoReset = TRUE
        DataUpdate:
          Activation:
            TimeStamp = TRUE
            Snippets = TRUE
        Recording:
          ActiveToInactive = FALSE
          AcknowledgedToUnacknowledged = FALSE
    [66]:
      Name = EventIDCode.6148
      Message = {$IAT/TrakError/Code.6148} Count: {&Cnt.6148} | {$IAT/TrakError/CheckLogBook}
      Behavior = UserDefined
        AutoReset = TRUE
        DataUpdate:
          Activation:
            TimeStamp = TRUE
            Snippets = TRUE
        Recording:
          ActiveToInactive = FALSE
          AcknowledgedToUnacknowledged = FALSE
    [67]:
      Name = EventIDCode.6149
      Message = {$IAT/TrakError/Code.6149} Count: {&Cnt.6149} | {$IAT/TrakError/CheckLogBook}
      Behavior = UserDefined
        AutoReset = TRUE
        DataUpdate:
          Activation:
            TimeStamp = TRUE
            Snippets = TRUE
        Recording:
          ActiveToInactive = FALSE
          AcknowledgedToUnacknowledged = FALSE
    [68]:
      Name = EventIDCode.6156
      Message = {$IAT/TrakError/Code.6156} Count: {&Cnt.6156} | {$IAT/TrakError/CheckLogBook}
      Behavior = UserDefined
        AutoReset = TRUE
        DataUpdate:
          Activation:
            TimeStamp = TRUE
            Snippets = TRUE
        Recording:
          ActiveToInactive = FALSE
          AcknowledgedToUnacknowledged = FALSE
    [69]:
      Name = EventIDCode.6157
      Message = {$IAT/TrakError/Code.6157} Count: {&Cnt.6157} | {$IAT/TrakError/CheckLogBook}
      Behavior = UserDefined
        AutoReset = TRUE
        DataUpdate:
          Activation:
            TimeStamp = TRUE
            Snippets = TRUE
        Recording:
          ActiveToInactive = FALSE
          AcknowledgedToUnacknowledged = FALSE
    [70]:
      Name = EventIDCode.6158
      Message = {$IAT/TrakError/Code.6158} Count: {&Cnt.6158} | {$IAT/TrakError/CheckLogBook}
      Behavior = UserDefined
        AutoReset = TRUE
        DataUpdate:
          Activation:
            TimeStamp = TRUE
            Snippets = TRUE
        Recording:
          ActiveToInactive = FALSE
          AcknowledgedToUnacknowledged = FALSE
    [71]:
      Name = EventIDCode.12288
      Message = {$IAT/TrakError/Code.12288} Count: {&Cnt.12288} | {$IAT/TrakError/CheckLogBook}
      Behavior = UserDefined
        AutoReset = TRUE
        DataUpdate:
          Activation:
            TimeStamp = TRUE
            Snippets = TRUE
        Recording:
          ActiveToInactive = FALSE
          AcknowledgedToUnacknowledged = FALSE
    [72]:
      Name = EventIDCode.12291
      Message = {$IAT/TrakError/Code.12291} Count: {&Cnt.12291} | {$IAT/TrakError/CheckLogBook}
      Behavior = UserDefined
        AutoReset = TRUE
        DataUpdate:
          Activation:
            TimeStamp = TRUE
            Snippets = TRUE
        Recording:
          ActiveToInactive = FALSE
          AcknowledgedToUnacknowledged = FALSE
    [73]:
      Name = EventIDCode.12293
      Message = {$IAT/TrakError/Code.12293} Count: {&Cnt.12293} | {$IAT/TrakError/CheckLogBook}
      Behavior = UserDefined
        AutoReset = TRUE
        DataUpdate:
          Activation:
            TimeStamp = TRUE
            Snippets = TRUE
        Recording:
          ActiveToInactive = FALSE
          AcknowledgedToUnacknowledged = FALSE
    [74]:
      Name = EventIDCode.12294
      Message = {$IAT/TrakError/Code.12294} Count: {&Cnt.12294} | {$IAT/TrakError/CheckLogBook}
      Behavior = UserDefined
        AutoReset = TRUE
        DataUpdate:
          Activation:
            TimeStamp = TRUE
            Snippets = TRUE
        Recording:
          ActiveToInactive = FALSE
          AcknowledgedToUnacknowledged = FALSE
    [75]:
      Name = EventIDCode.12295
      Message = {$IAT/TrakError/Code.12295} Count: {&Cnt.12295} | {$IAT/TrakError/CheckLogBook}
      Behavior = UserDefined
        AutoReset = TRUE
        DataUpdate:
          Activation:
            TimeStamp = TRUE
            Snippets = TRUE
        Recording:
          ActiveToInactive = FALSE
          AcknowledgedToUnacknowledged = FALSE
    [76]:
      Name = EventIDCode.12296
      Message = {$IAT/TrakError/Code.12296} Count: {&Cnt.12296} | {$IAT/TrakError/CheckLogBook}
      Behavior = UserDefined
        AutoReset = TRUE
        DataUpdate:
          Activation:
            TimeStamp = TRUE
            Snippets = TRUE
        Recording:
          ActiveToInactive = FALSE
          AcknowledgedToUnacknowledged = FALSE
    [77]:
      Name = EventIDCode.12297
      Message = {$IAT/TrakError/Code.12297} Count: {&Cnt.12297} | {$IAT/TrakError/CheckLogBook}
      Behavior = UserDefined
        AutoReset = TRUE
        DataUpdate:
          Activation:
            TimeStamp = TRUE
            Snippets = TRUE
        Recording:
          ActiveToInactive = FALSE
          AcknowledgedToUnacknowledged = FALSE
    [78]:
      Name = EventIDCode.12298
      Message = {$IAT/TrakError/Code.12298} Count: {&Cnt.12298} | {$IAT/TrakError/CheckLogBook}
      Behavior = UserDefined
        AutoReset = TRUE
        DataUpdate:
          Activation:
            TimeStamp = TRUE
            Snippets = TRUE
        Recording:
          ActiveToInactive = FALSE
          AcknowledgedToUnacknowledged = FALSE
    [79]:
      Name = EventIDCode.12299
      Message = {$IAT/TrakError/Code.12299} Count: {&Cnt.12299} | {$IAT/TrakError/CheckLogBook}
      Behavior = UserDefined
        AutoReset = TRUE
        DataUpdate:
          Activation:
            TimeStamp = TRUE
            Snippets = TRUE
        Recording:
          ActiveToInactive = FALSE
          AcknowledgedToUnacknowledged = FALSE
    [80]:
      Name = EventIDCode.12300
      Message = {$IAT/TrakError/Code.12300} Count: {&Cnt.12300} | {$IAT/TrakError/CheckLogBook}
      Behavior = UserDefined
        AutoReset = TRUE
        DataUpdate:
          Activation:
            TimeStamp = TRUE
            Snippets = TRUE
        Recording:
          ActiveToInactive = FALSE
          AcknowledgedToUnacknowledged = FALSE
    [81]:
      Name = EventIDCode.12301
      Message = {$IAT/TrakError/Code.12301} Count: {&Cnt.12301} | {$IAT/TrakError/CheckLogBook}
      Behavior = UserDefined
        AutoReset = TRUE
        DataUpdate:
          Activation:
            TimeStamp = TRUE
            Snippets = TRUE
        Recording:
          ActiveToInactive = FALSE
          AcknowledgedToUnacknowledged = FALSE
    [82]:
      Name = EventIDCode.12302
      Message = {$IAT/TrakError/Code.12302} Count: {&Cnt.12302} | {$IAT/TrakError/CheckLogBook}
      Behavior = UserDefined
        AutoReset = TRUE
        DataUpdate:
          Activation:
            TimeStamp = TRUE
            Snippets = TRUE
        Recording:
          ActiveToInactive = FALSE
          AcknowledgedToUnacknowledged = FALSE
    [83]:
      Name = EventIDCode.12303
      Message = {$IAT/TrakError/Code.12303} Count: {&Cnt.12303} | {$IAT/TrakError/CheckLogBook}
      Behavior = UserDefined
        AutoReset = TRUE
        DataUpdate:
          Activation:
            TimeStamp = TRUE
            Snippets = TRUE
        Recording:
          ActiveToInactive = FALSE
          AcknowledgedToUnacknowledged = FALSE
    [84]:
      Name = EventIDCode.12304
      Message = {$IAT/TrakError/Code.12304} Count: {&Cnt.12304} | {$IAT/TrakError/CheckLogBook}
      Behavior = UserDefined
        AutoReset = TRUE
        DataUpdate:
          Activation:
            TimeStamp = TRUE
            Snippets = TRUE
        Recording:
          ActiveToInactive = FALSE
          AcknowledgedToUnacknowledged = FALSE
    [85]:
      Name = EventIDCode.12305
      Message = {$IAT/TrakError/Code.12305} Count: {&Cnt.12305} | {$IAT/TrakError/CheckLogBook}
      Behavior = UserDefined
        AutoReset = TRUE
        DataUpdate:
          Activation:
            TimeStamp = TRUE
            Snippets = TRUE
        Recording:
          ActiveToInactive = FALSE
          AcknowledgedToUnacknowledged = FALSE
    [86]:
      Name = EventIDCode.12307
      Message = {$IAT/TrakError/Code.12307} Count: {&Cnt.12307} | {$IAT/TrakError/CheckLogBook}
      Behavior = UserDefined
        AutoReset = TRUE
        DataUpdate:
          Activation:
            TimeStamp = TRUE
            Snippets = TRUE
        Recording:
          ActiveToInactive = FALSE
          AcknowledgedToUnacknowledged = FALSE
    [87]:
      Name = EventIDCode.12312
      Message = {$IAT/TrakError/Code.12312} Count: {&Cnt.12312} | {$IAT/TrakError/CheckLogBook}
      Behavior = UserDefined
        AutoReset = TRUE
        DataUpdate:
          Activation:
            TimeStamp = TRUE
            Snippets = TRUE
        Recording:
          ActiveToInactive = FALSE
          AcknowledgedToUnacknowledged = FALSE
    [88]:
      Name = EventIDCode.12313
      Message = {$IAT/TrakError/Code.12313} Count: {&Cnt.12313} | {$IAT/TrakError/CheckLogBook}
      Behavior = UserDefined
        AutoReset = TRUE
        DataUpdate:
          Activation:
            TimeStamp = TRUE
            Snippets = TRUE
        Recording:
          ActiveToInactive = FALSE
          AcknowledgedToUnacknowledged = FALSE
    [89]:
      Name = EventIDCode.12314
      Message = {$IAT/TrakError/Code.12314} Count: {&Cnt.12314} | {$IAT/TrakError/CheckLogBook}
      Behavior = UserDefined
        AutoReset = TRUE
        DataUpdate:
          Activation:
            TimeStamp = TRUE
            Snippets = TRUE
        Recording:
          ActiveToInactive = FALSE
          AcknowledgedToUnacknowledged = FALSE
    [90]:
      Name = EventIDCode.12315
      Message = {$IAT/TrakError/Code.12315} Count: {&Cnt.12315} | {$IAT/TrakError/CheckLogBook}
      Behavior = UserDefined
        AutoReset = TRUE
        DataUpdate:
          Activation:
            TimeStamp = TRUE
            Snippets = TRUE
        Recording:
          ActiveToInactive = FALSE
          AcknowledgedToUnacknowledged = FALSE
    [91]:
      Name = EventIDCode.12316
      Message = {$IAT/TrakError/Code.12316} Count: {&Cnt.12316} | {$IAT/TrakError/CheckLogBook}
      Behavior = UserDefined
        AutoReset = TRUE
        DataUpdate:
          Activation:
            TimeStamp = TRUE
            Snippets = TRUE
        Recording:
          ActiveToInactive = FALSE
          AcknowledgedToUnacknowledged = FALSE
    [92]:
      Name = EventIDCode.12317
      Message = {$IAT/TrakError/Code.12317} Count: {&Cnt.12317} | {$IAT/TrakError/CheckLogBook}
      Behavior = UserDefined
        AutoReset = TRUE
        DataUpdate:
          Activation:
            TimeStamp = TRUE
            Snippets = TRUE
        Recording:
          ActiveToInactive = FALSE
          AcknowledgedToUnacknowledged = FALSE
    [93]:
      Name = EventIDCode.12320
      Message = {$IAT/TrakError/Code.12320} Count: {&Cnt.12320} | {$IAT/TrakError/CheckLogBook}
      Behavior = UserDefined
        AutoReset = TRUE
        DataUpdate:
          Activation:
            TimeStamp = TRUE
            Snippets = TRUE
        Recording:
          ActiveToInactive = FALSE
          AcknowledgedToUnacknowledged = FALSE
    [94]:
      Name = EventIDCode.12322
      Message = {$IAT/TrakError/Code.12322} Count: {&Cnt.12322} | {$IAT/TrakError/CheckLogBook}
      Behavior = UserDefined
        AutoReset = TRUE
        DataUpdate:
          Activation:
            TimeStamp = TRUE
            Snippets = TRUE
        Recording:
          ActiveToInactive = FALSE
          AcknowledgedToUnacknowledged = FALSE
    [95]:
      Name = EventIDCode.12323
      Message = {$IAT/TrakError/Code.12323} Count: {&Cnt.12323} | {$IAT/TrakError/CheckLogBook}
      Behavior = UserDefined
        AutoReset = TRUE
        DataUpdate:
          Activation:
            TimeStamp = TRUE
            Snippets = TRUE
        Recording:
          ActiveToInactive = FALSE
          AcknowledgedToUnacknowledged = FALSE
    [96]:
      Name = EventIDCode.12328
      Message = {$IAT/TrakError/Code.12328} Count: {&Cnt.12328} | {$IAT/TrakError/CheckLogBook}
      Behavior = UserDefined
        AutoReset = TRUE
        DataUpdate:
          Activation:
            TimeStamp = TRUE
            Snippets = TRUE
        Recording:
          ActiveToInactive = FALSE
          AcknowledgedToUnacknowledged = FALSE
    [97]:
      Name = EventIDCode.12330
      Message = {$IAT/TrakError/Code.12330} Count: {&Cnt.12330} | {$IAT/TrakError/CheckLogBook}
      Behavior = UserDefined
        AutoReset = TRUE
        DataUpdate:
          Activation:
            TimeStamp = TRUE
            Snippets = TRUE
        Recording:
          ActiveToInactive = FALSE
          AcknowledgedToUnacknowledged = FALSE
    [98]:
      Name = EventIDCode.12331
      Message = {$IAT/TrakError/Code.12331} Count: {&Cnt.12331} | {$IAT/TrakError/CheckLogBook}
      Behavior = UserDefined
        AutoReset = TRUE
        DataUpdate:
          Activation:
            TimeStamp = TRUE
            Snippets = TRUE
        Recording:
          ActiveToInactive = FALSE
          AcknowledgedToUnacknowledged = FALSE
    [99]:
      Name = EventIDCode.12333
      Message = {$IAT/TrakError/Code.12333} Count: {&Cnt.12333} | {$IAT/TrakError/CheckLogBook}
      Behavior = UserDefined
        AutoReset = TRUE
        DataUpdate:
          Activation:
            TimeStamp = TRUE
            Snippets = TRUE
        Recording:
          ActiveToInactive = FALSE
          AcknowledgedToUnacknowledged = FALSE
    [100]:
      Name = EventIDCode.12334
      Message = {$IAT/TrakError/Code.12334} Count: {&Cnt.12334} | {$IAT/TrakError/CheckLogBook}
      Behavior = UserDefined
        AutoReset = TRUE
        DataUpdate:
          Activation:
            TimeStamp = TRUE
            Snippets = TRUE
        Recording:
          ActiveToInactive = FALSE
          AcknowledgedToUnacknowledged = FALSE
    [101]:
      Name = EventIDCode.12335
      Message = {$IAT/TrakError/Code.12335} Count: {&Cnt.12335} | {$IAT/TrakError/CheckLogBook}
      Behavior = UserDefined
        AutoReset = TRUE
        DataUpdate:
          Activation:
            TimeStamp = TRUE
            Snippets = TRUE
        Recording:
          ActiveToInactive = FALSE
          AcknowledgedToUnacknowledged = FALSE
    [102]:
      Name = EventIDCode.12336
      Message = {$IAT/TrakError/Code.12336} Count: {&Cnt.12336} | {$IAT/TrakError/CheckLogBook}
      Behavior = UserDefined
        AutoReset = TRUE
        DataUpdate:
          Activation:
            TimeStamp = TRUE
            Snippets = TRUE
        Recording:
          ActiveToInactive = FALSE
          AcknowledgedToUnacknowledged = FALSE
    [103]:
      Name = EventIDCode.12337
      Message = {$IAT/TrakError/Code.12337} Count: {&Cnt.12337} | {$IAT/TrakError/CheckLogBook}
      Behavior = UserDefined
        AutoReset = TRUE
        DataUpdate:
          Activation:
            TimeStamp = TRUE
            Snippets = TRUE
        Recording:
          ActiveToInactive = FALSE
          AcknowledgedToUnacknowledged = FALSE
    [104]:
      Name = EventIDCode.12338
      Message = {$IAT/TrakError/Code.12338} Count: {&Cnt.12338} | {$IAT/TrakError/CheckLogBook}
      Behavior = UserDefined
        AutoReset = TRUE
        DataUpdate:
          Activation:
            TimeStamp = TRUE
            Snippets = TRUE
        Recording:
          ActiveToInactive = FALSE
          AcknowledgedToUnacknowledged = FALSE
    [105]:
      Name = EventIDCode.12340
      Message = {$IAT/TrakError/Code.12340} Count: {&Cnt.12340} | {$IAT/TrakError/CheckLogBook}
      Behavior = UserDefined
        AutoReset = TRUE
        DataUpdate:
          Activation:
            TimeStamp = TRUE
            Snippets = TRUE
        Recording:
          ActiveToInactive = FALSE
          AcknowledgedToUnacknowledged = FALSE
    [106]:
      Name = EventIDCode.12341
      Message = {$IAT/TrakError/Code.12341} Count: {&Cnt.12341} | {$IAT/TrakError/CheckLogBook}
      Behavior = UserDefined
        AutoReset = TRUE
        DataUpdate:
          Activation:
            TimeStamp = TRUE
            Snippets = TRUE
        Recording:
          ActiveToInactive = FALSE
          AcknowledgedToUnacknowledged = FALSE
    [107]:
      Name = EventIDCode.12342
      Message = {$IAT/TrakError/Code.12342} Count: {&Cnt.12342} | {$IAT/TrakError/CheckLogBook}
      Behavior = UserDefined
        AutoReset = TRUE
        DataUpdate:
          Activation:
            TimeStamp = TRUE
            Snippets = TRUE
        Recording:
          ActiveToInactive = FALSE
          AcknowledgedToUnacknowledged = FALSE
    [108]:
      Name = EventIDCode.12343
      Message = {$IAT/TrakError/Code.12343} Count: {&Cnt.12343} | {$IAT/TrakError/CheckLogBook}
      Behavior = UserDefined
        AutoReset = TRUE
        DataUpdate:
          Activation:
            TimeStamp = TRUE
            Snippets = TRUE
        Recording:
          ActiveToInactive = FALSE
          AcknowledgedToUnacknowledged = FALSE
    [109]:
      Name = EventIDCode.12344
      Message = {$IAT/TrakError/Code.12344} Count: {&Cnt.12344} | {$IAT/TrakError/CheckLogBook}
      Behavior = UserDefined
        AutoReset = TRUE
        DataUpdate:
          Activation:
            TimeStamp = TRUE
            Snippets = TRUE
        Recording:
          ActiveToInactive = FALSE
          AcknowledgedToUnacknowledged = FALSE
    [110]:
      Name = EventIDCode.12345
      Message = {$IAT/TrakError/Code.12345} Count: {&Cnt.12345} | {$IAT/TrakError/CheckLogBook}
      Behavior = UserDefined
        AutoReset = TRUE
        DataUpdate:
          Activation:
            TimeStamp = TRUE
            Snippets = TRUE
        Recording:
          ActiveToInactive = FALSE
          AcknowledgedToUnacknowledged = FALSE
    [111]:
      Name = EventIDCode.12346
      Message = {$IAT/TrakError/Code.12346} Count: {&Cnt.12346} | {$IAT/TrakError/CheckLogBook}
      Behavior = UserDefined
        AutoReset = TRUE
        DataUpdate:
          Activation:
            TimeStamp = TRUE
            Snippets = TRUE
        Recording:
          ActiveToInactive = FALSE
          AcknowledgedToUnacknowledged = FALSE
    [112]:
      Name = EventIDCode.12347
      Message = {$IAT/TrakError/Code.12347} Count: {&Cnt.12347} | {$IAT/TrakError/CheckLogBook}
      Behavior = UserDefined
        AutoReset = TRUE
        DataUpdate:
          Activation:
            TimeStamp = TRUE
            Snippets = TRUE
        Recording:
          ActiveToInactive = FALSE
          AcknowledgedToUnacknowledged = FALSE
    [113]:
      Name = EventIDCode.12348
      Message = {$IAT/TrakError/Code.12348} Count: {&Cnt.12348} | {$IAT/TrakError/CheckLogBook}
      Behavior = UserDefined
        AutoReset = TRUE
        DataUpdate:
          Activation:
            TimeStamp = TRUE
            Snippets = TRUE
        Recording:
          ActiveToInactive = FALSE
          AcknowledgedToUnacknowledged = FALSE
    [114]:
      Name = EventIDCode.4007
      Message = {$IAT/TrakError/Code.4007} Count: {&Cnt.4007} | {$IAT/TrakError/CheckLogBook}
      Behavior = UserDefined
        AutoReset = TRUE
        DataUpdate:
          Activation:
            TimeStamp = TRUE
            Snippets = TRUE
        Recording:
          ActiveToInactive = FALSE
          AcknowledgedToUnacknowledged = FALSE
    [115]:
      Name = EventIDCode.7230
      Message = {$IAT/TrakError/Code.7230} Count: {&Cnt.7230} | {$IAT/TrakError/CheckLogBook}
      Behavior = UserDefined
        AutoReset = TRUE
        DataUpdate:
          Activation:
            TimeStamp = TRUE
            Snippets = TRUE
        Recording:
          ActiveToInactive = FALSE
          AcknowledgedToUnacknowledged = FALSE
    [116]:
      Name = EventIDCode.4005
      Message = {$IAT/TrakError/Code.4005} Count: {&Cnt.4005} | {$IAT/TrakError/CheckLogBook}
      Behavior = UserDefined
        AutoReset = TRUE
        DataUpdate:
          Activation:
            TimeStamp = TRUE
            Snippets = TRUE
        Recording:
          ActiveToInactive = FALSE
          AcknowledgedToUnacknowledged = FALSE
    [117]:
      Name = EventIDCode.4098
      Message = {$IAT/TrakError/Code.4098} Count: {&Cnt.4098} | {$IAT/TrakError/CheckLogBook}
      Behavior = UserDefined
        AutoReset = TRUE
        DataUpdate:
          Activation:
            TimeStamp = TRUE
            Snippets = TRUE
        Recording:
          ActiveToInactive = FALSE
          AcknowledgedToUnacknowledged = FALSE
    [118]:
      Name = EventIDCode.9106
      Message = {$IAT/TrakError/Code.9106} Count: {&Cnt.9106} | {$IAT/TrakError/CheckLogBook}
      Behavior = UserDefined
        AutoReset = TRUE
        DataUpdate:
          Activation:
            TimeStamp = TRUE
            Snippets = TRUE
        Recording:
          ActiveToInactive = FALSE
          AcknowledgedToUnacknowledged = FALSE
    [119]:
      Name = EventIDCode.xxxx
      Message = {$IAT/TrakError/Code.xxxx} Count: {&Cnt.xxxx} | {$IAT/TrakError/CheckLogBook}
      Behavior = UserDefined
        AutoReset = TRUE
        DataUpdate:
          Activation:
            TimeStamp = TRUE
            Snippets = TRUE
        Recording:
          ActiveToInactive = FALSE
          AcknowledgedToUnacknowledged = FALSE
  mapp.AlarmX.Core.Snippets:
    [0]:
      Key = ModuleName
      Value:
        PV = Diag::ModuleName
    [1]:
      Key = Cnt.1
      Value:
        PV = Diag::Logbook:AlarmCount[0]
    [2]:
      Key = Cnt.2
      Value:
        PV = Diag::Logbook:AlarmCount[1]
    [3]:
      Key = Cnt.7
      Value:
        PV = Diag::Logbook:AlarmCount[2]
    [4]:
      Key = Cnt.2048
      Value:
        PV = Diag::Logbook:AlarmCount[3]
    [5]:
      Key = Cnt.2049
      Value:
        PV = Diag::Logbook:AlarmCount[4]
    [6]:
      Key = Cnt.2050
      Value:
        PV = Diag::Logbook:AlarmCount[5]
    [7]:
      Key = Cnt.2051
      Value:
        PV = Diag::Logbook:AlarmCount[6]
    [8]:
      Key = Cnt.2052
      Value:
        PV = Diag::Logbook:AlarmCount[7]
    [9]:
      Key = Cnt.2053
      Value:
        PV = Diag::Logbook:AlarmCount[8]
    [10]:
      Key = Cnt.2054
      Value:
        PV = Diag::Logbook:AlarmCount[9]
    [11]:
      Key = Cnt.2055
      Value:
        PV = Diag::Logbook:AlarmCount[10]
    [12]:
      Key = Cnt.2056
      Value:
        PV = Diag::Logbook:AlarmCount[11]
    [13]:
      Key = Cnt.2057
      Value:
        PV = Diag::Logbook:AlarmCount[12]
    [14]:
      Key = Cnt.2058
      Value:
        PV = Diag::Logbook:AlarmCount[13]
    [15]:
      Key = Cnt.2060
      Value:
        PV = Diag::Logbook:AlarmCount[14]
    [16]:
      Key = Cnt.2061
      Value:
        PV = Diag::Logbook:AlarmCount[15]
    [17]:
      Key = Cnt.2063
      Value:
        PV = Diag::Logbook:AlarmCount[16]
    [18]:
      Key = Cnt.2064
      Value:
        PV = Diag::Logbook:AlarmCount[17]
    [19]:
      Key = Cnt.2066
      Value:
        PV = Diag::Logbook:AlarmCount[18]
    [20]:
      Key = Cnt.2067
      Value:
        PV = Diag::Logbook:AlarmCount[19]
    [21]:
      Key = Cnt.2068
      Value:
        PV = Diag::Logbook:AlarmCount[20]
    [22]:
      Key = Cnt.2069
      Value:
        PV = Diag::Logbook:AlarmCount[21]
    [23]:
      Key = Cnt.2070
      Value:
        PV = Diag::Logbook:AlarmCount[22]
    [24]:
      Key = Cnt.2071
      Value:
        PV = Diag::Logbook:AlarmCount[23]
    [25]:
      Key = Cnt.2074
      Value:
        PV = Diag::Logbook:AlarmCount[24]
    [26]:
      Key = Cnt.2077
      Value:
        PV = Diag::Logbook:AlarmCount[25]
    [27]:
      Key = Cnt.2080
      Value:
        PV = Diag::Logbook:AlarmCount[26]
    [28]:
      Key = Cnt.2082
      Value:
        PV = Diag::Logbook:AlarmCount[27]
    [29]:
      Key = Cnt.2083
      Value:
        PV = Diag::Logbook:AlarmCount[28]
    [30]:
      Key = Cnt.2084
      Value:
        PV = Diag::Logbook:AlarmCount[29]
    [31]:
      Key = Cnt.2085
      Value:
        PV = Diag::Logbook:AlarmCount[30]
    [32]:
      Key = Cnt.2090
      Value:
        PV = Diag::Logbook:AlarmCount[31]
    [33]:
      Key = Cnt.2091
      Value:
        PV = Diag::Logbook:AlarmCount[32]
    [34]:
      Key = Cnt.2092
      Value:
        PV = Diag::Logbook:AlarmCount[33]
    [35]:
      Key = Cnt.2093
      Value:
        PV = Diag::Logbook:AlarmCount[34]
    [36]:
      Key = Cnt.2094
      Value:
        PV = Diag::Logbook:AlarmCount[35]
    [37]:
      Key = Cnt.2095
      Value:
        PV = Diag::Logbook:AlarmCount[36]
    [38]:
      Key = Cnt.2097
      Value:
        PV = Diag::Logbook:AlarmCount[37]
    [39]:
      Key = Cnt.2098
      Value:
        PV = Diag::Logbook:AlarmCount[38]
    [40]:
      Key = Cnt.2099
      Value:
        PV = Diag::Logbook:AlarmCount[39]
    [41]:
      Key = Cnt.2100
      Value:
        PV = Diag::Logbook:AlarmCount[40]
    [42]:
      Key = Cnt.2101
      Value:
        PV = Diag::Logbook:AlarmCount[41]
    [43]:
      Key = Cnt.2102
      Value:
        PV = Diag::Logbook:AlarmCount[42]
    [44]:
      Key = Cnt.2103
      Value:
        PV = Diag::Logbook:AlarmCount[43]
    [45]:
      Key = Cnt.2104
      Value:
        PV = Diag::Logbook:AlarmCount[44]
    [46]:
      Key = Cnt.2105
      Value:
        PV = Diag::Logbook:AlarmCount[45]
    [47]:
      Key = Cnt.2106
      Value:
        PV = Diag::Logbook:AlarmCount[46]
    [48]:
      Key = Cnt.2107
      Value:
        PV = Diag::Logbook:AlarmCount[47]
    [49]:
      Key = Cnt.2108
      Value:
        PV = Diag::Logbook:AlarmCount[48]
    [50]:
      Key = Cnt.2109
      Value:
        PV = Diag::Logbook:AlarmCount[49]
    [51]:
      Key = Cnt.2110
      Value:
        PV = Diag::Logbook:AlarmCount[50]
    [52]:
      Key = Cnt.2111
      Value:
        PV = Diag::Logbook:AlarmCount[51]
    [53]:
      Key = Cnt.2112
      Value:
        PV = Diag::Logbook:AlarmCount[52]
    [54]:
      Key = Cnt.4096
      Value:
        PV = Diag::Logbook:AlarmCount[53]
    [55]:
      Key = Cnt.4097
      Value:
        PV = Diag::Logbook:AlarmCount[54]
    [56]:
      Key = Cnt.4101
      Value:
        PV = Diag::Logbook:AlarmCount[55]
    [57]:
      Key = Cnt.4102
      Value:
        PV = Diag::Logbook:AlarmCount[56]
    [58]:
      Key = Cnt.6144
      Value:
        PV = Diag::Logbook:AlarmCount[57]
    [59]:
      Key = Cnt.6165
      Value:
        PV = Diag::Logbook:AlarmCount[58]
    [60]:
      Key = Cnt.6148
      Value:
        PV = Diag::Logbook:AlarmCount[59]
    [61]:
      Key = Cnt.6149
      Value:
        PV = Diag::Logbook:AlarmCount[60]
    [62]:
      Key = Cnt.6156
      Value:
        PV = Diag::Logbook:AlarmCount[61]
    [63]:
      Key = Cnt.6157
      Value:
        PV = Diag::Logbook:AlarmCount[62]
    [64]:
      Key = Cnt.6158
      Value:
        PV = Diag::Logbook:AlarmCount[63]
    [65]:
      Key = Cnt.12288
      Value:
        PV = Diag::Logbook:AlarmCount[64]
    [66]:
      Key = Cnt.12291
      Value:
        PV = Diag::Logbook:AlarmCount[65]
    [67]:
      Key = Cnt.12293
      Value:
        PV = Diag::Logbook:AlarmCount[66]
    [68]:
      Key = Cnt.12294
      Value:
        PV = Diag::Logbook:AlarmCount[67]
    [69]:
      Key = Cnt.12295
      Value:
        PV = Diag::Logbook:AlarmCount[68]
    [70]:
      Key = Cnt.12296
      Value:
        PV = Diag::Logbook:AlarmCount[69]
    [71]:
      Key = Cnt.12297
      Value:
        PV = Diag::Logbook:AlarmCount[70]
    [72]:
      Key = Cnt.12298
      Value:
        PV = Diag::Logbook:AlarmCount[71]
    [73]:
      Key = Cnt.12299
      Value:
        PV = Diag::Logbook:AlarmCount[72]
    [74]:
      Key = Cnt.12300
      Value:
        PV = Diag::Logbook:AlarmCount[73]
    [75]:
      Key = Cnt.12301
      Value:
        PV = Diag::Logbook:AlarmCount[74]
    [76]:
      Key = Cnt.12302
      Value:
        PV = Diag::Logbook:AlarmCount[75]
    [77]:
      Key = Cnt.12303
      Value:
        PV = Diag::Logbook:AlarmCount[76]
    [78]:
      Key = Cnt.12304
      Value:
        PV = Diag::Logbook:AlarmCount[77]
    [79]:
      Key = Cnt.12305
      Value:
        PV = Diag::Logbook:AlarmCount[78]
    [80]:
      Key = Cnt.12307
      Value:
        PV = Diag::Logbook:AlarmCount[79]
    [81]:
      Key = Cnt.12312
      Value:
        PV = Diag::Logbook:AlarmCount[80]
    [82]:
      Key = Cnt.12313
      Value:
        PV = Diag::Logbook:AlarmCount[81]
    [83]:
      Key = Cnt.12314
      Value:
        PV = Diag::Logbook:AlarmCount[82]
    [84]:
      Key = Cnt.12315
      Value:
        PV = Diag::Logbook:AlarmCount[83]
    [85]:
      Key = Cnt.12316
      Value:
        PV = Diag::Logbook:AlarmCount[84]
    [86]:
      Key = Cnt.12317
      Value:
        PV = Diag::Logbook:AlarmCount[85]
    [87]:
      Key = Cnt.12320
      Value:
        PV = Diag::Logbook:AlarmCount[86]
    [88]:
      Key = Cnt.12322
      Value:
        PV = Diag::Logbook:AlarmCount[87]
    [89]:
      Key = Cnt.12323
      Value:
        PV = Diag::Logbook:AlarmCount[88]
    [90]:
      Key = Cnt.12328
      Value:
        PV = Diag::Logbook:AlarmCount[89]
    [91]:
      Key = Cnt.12330
      Value:
        PV = Diag::Logbook:AlarmCount[90]
    [92]:
      Key = Cnt.12331
      Value:
        PV = Diag::Logbook:AlarmCount[91]
    [93]:
      Key = Cnt.12333
      Value:
        PV = Diag::Logbook:AlarmCount[92]
    [94]:
      Key = Cnt.12334
      Value:
        PV = Diag::Logbook:AlarmCount[93]
    [95]:
      Key = Cnt.12335
      Value:
        PV = Diag::Logbook:AlarmCount[94]
    [96]:
      Key = Cnt.12336
      Value:
        PV = Diag::Logbook:AlarmCount[95]
    [97]:
      Key = Cnt.12337
      Value:
        PV = Diag::Logbook:AlarmCount[96]
    [98]:
      Key = Cnt.12338
      Value:
        PV = Diag::Logbook:AlarmCount[97]
    [99]:
      Key = Cnt.12340
      Value:
        PV = Diag::Logbook:AlarmCount[98]
    [100]:
      Key = Cnt.12341
      Value:
        PV = Diag::Logbook:AlarmCount[99]
    [101]:
      Key = Cnt.12342
      Value:
        PV = Diag::Logbook:AlarmCount[100]
    [102]:
      Key = Cnt.12343
      Value:
        PV = Diag::Logbook:AlarmCount[101]
    [103]:
      Key = Cnt.12344
      Value:
        PV = Diag::Logbook:AlarmCount[102]
    [104]:
      Key = Cnt.12345
      Value:
        PV = Diag::Logbook:AlarmCount[103]
    [105]:
      Key = Cnt.12346
      Value:
        PV = Diag::Logbook:AlarmCount[104]
    [106]:
      Key = Cnt.12347
      Value:
        PV = Diag::Logbook:AlarmCount[105]
    [107]:
      Key = Cnt.12348
      Value:
        PV = Diag::Logbook:AlarmCount[106]
    [108]:
      Key = Cnt.4007
      Value:
        PV = Diag::Logbook:AlarmCount[107]
    [109]:
      Key = Cnt.7230
      Value:
        PV = Diag::Logbook:AlarmCount[108]
    [110]:
      Key = Cnt.4005
      Value:
        PV = Diag::Logbook:AlarmCount[109]
    [111]:
      Key = Cnt.4098
      Value:
        PV = Diag::Logbook:AlarmCount[110]
    [112]:
      Key = Cnt.9106
      Value:
        PV = Diag::Logbook:AlarmCount[111]
  mapp.AlarmX.Core.Categories:
    [0]:
      Name = Information
      SourceProperty:
        Severity = 0..99
    [1]:
      Name = Warning
      SourceProperty:
        Severity = 100..199
    [2]:
      Name = Alarm
      SourceProperty:
        Severity = 1000..1199
```

### DiagAUD.mpaudittrail - PC/Diag/mappServices/DiagAUD.mpaudittrail
```
Element gAuditTrail_DiagModule (Type=mpaudittrail)
  Audit:
    Events:
      [0] = 18
    TextSource:
      OutputFormat = {&typ} | {&msg} | {&cmt}
  Alarms = MpAlarmX
```

### DiagREC.mprecipexml - PC/Diag/mappServices/DiagREC.mprecipexml
```
Element gRecipeXml_DiagModule (Type=mprecipexml)
  Alarms = MpAlarmX
```

### EM12CFG.mprecipexml - PC/EM1/EM12/mappServices/EM12CFG.mprecipexml
```
Element gRecipeXml_2 (Type=mprecipexml)
```

### TrakALM.mpalarmxcore - PC/EM1/TrakModule/mappServices/TrakALM.mpalarmxcore
```
Element gAlarmXCore_1 (Type=mpalarmxcore)
```

### TrakCFG.mprecipexml - PC/EM1/TrakModule/mappServices/TrakCFG.mprecipexml
```
Element gRecipeXml_1 (Type=mprecipexml)
```

### TrakPML.mppackmlmodule - PC/EM1/TrakModule/mappServices/TrakPML.mppackmlmodule
```
Element gTrakModule (Type=mppackmlmodule)
  Module:
    Name = TrakAssembly
    Parent:
      Parent = gMainModule
      Activation = 1
```

### SubMod1.vvm - PC/EM12/SubMod1.vvm
```iecst
VAR_CONFIG
	Cyclic#1.::gMainModule AT %Q.EM12::ModuleInterface.MainPml; (*Insert your comment here...*)
END_VAR
```

### EM12ALM.mpalarmxcore - PC/EM12/mappServices/EM12ALM.mpalarmxcore
```
Element gAlarmXCore_2 (Type=mpalarmxcore)
  mapp.AlarmX.Core:
    Mapping:
      [0]:
        Alarm = Inf*
        [0] = Aggregate
          Name = TrakModuleInfo
      [1]:
        Alarm = Warn*
        [0] = Aggregate
          Name = TrakModuleWarning
        [1]
      [2]:
        Alarm = Alrm*
        [0] = Aggregate
          Name = TrakModuleAlarm
    Default:
      [0] = Remain
  mapp.AlarmX.Core.Categories:
    [0]:
      Name = Information
      SourceProperty:
        Severity = 0..99
    [1]:
      Name = Warning
      SourceProperty:
        Severity = 100..199
    [2]:
      Name = Alarm
      SourceProperty:
        Severity = 1000..1199
```

### EM12PML.mppackmlmodule - PC/EM12/mappServices/EM12PML.mppackmlmodule
```
Element gPackMLModule (Type=mppackmlmodule)
  Module:
    Parent:
      Parent = gMainModule
      Activation = 0
```

### EM2.vvm - PC/EM2/EM2.vvm
```iecst
VAR_CONFIG
	Cyclic#1.::gMainModule AT %Q.EM2::ModuleInterface.MainPml; (*Insert your comment here...*)
	Cyclic#1.EM2::gAlarmXCore_EM2 AT %Q.EM2::ModuleInterface.AlarmCore; (*Insert your comment here...*)
	EM2::gRecipeXml_EM2 AT %Q.EM2::ModuleInterface.RecipeCore; (*Insert your comment here...*)
	EM2::gPackMLModule_EM2 AT %Q.EM2::ModuleInterface.ModulePml; (*Insert your comment here...*)
END_VAR
```

### EM2ALM.mpalarmxcore - PC/EM2/mappServices/EM2ALM.mpalarmxcore
```
Element gAlarmXCore_EM2 (Type=mpalarmxcore)
  mapp.AlarmX.Core:
    Mapping:
      [0]:
        Alarm = Inf*
        [0] = Aggregate
          Name = ModuleInfo
      [1]:
        Alarm = Warn*
        [0] = Aggregate
          Name = ModuleWarning
        [1]
      [2]:
        Alarm = Alrm*
        [0] = Aggregate
          Name = ModuleAlarm
    Default:
      [0] = Remain
  mapp.AlarmX.Core.Configuration:
    [0]:
      Name = Inf_ModuleOperation
      Message = {$AppModule/Operation.Info}
      Severity = 0
      Behavior = DiscreteValueMonitoring
        Monitoring:
          MonitoredPV = EM2::OperationInformation
          TriggerValues:
            [0] = TRUE
    [1]:
      Name = Warn_ModuleOperation
      Message = {$AppModule/Operation.Warning}
      Severity = 0
      Behavior = DiscreteValueMonitoring
        Monitoring:
          MonitoredPV = EM2::OperationWarning
          TriggerValues:
            [0] = TRUE
    [2]:
      Name = Alrm_ModuleOperation
      Message = {$AppModule/Operation.Alarm}
      Severity = 0
      Behavior = DiscreteValueMonitoring
        Monitoring:
          MonitoredPV = EM2::OperationAlarm
          TriggerValues:
            [0] = TRUE
    [3]:
      Name = Inf_ModuleConfig
      Message = {$AppModule/Configuration.Info}
      Severity = 0
      Behavior = DiscreteValueMonitoring
        Monitoring:
          MonitoredPV = EM2::ConfigInformation
          TriggerValues:
            [0] = TRUE
    [4]:
      Name = Warn_ModuleConfig
      Message = {$AppModule/Configuration.Warning}
      Severity = 0
      Behavior = DiscreteValueMonitoring
        Monitoring:
          MonitoredPV = EM2::ConfigWarning
          TriggerValues:
            [0] = TRUE
    [5]:
      Name = Alrm_ModuleConfig
      Message = {$AppModule/Configuration.Alarm}
      Severity = 0
      Behavior = DiscreteValueMonitoring
        Monitoring:
          MonitoredPV = EM2::ConfigAlarm
          TriggerValues:
            [0] = TRUE
    [6]:
      Name = Inf_ModuleRecovery
      Message = {$AppModule/Recovery.Info}
      Severity = 0
      Behavior = DiscreteValueMonitoring
        Monitoring:
          MonitoredPV = EM2::RecoveryInformation
          TriggerValues:
            [0] = TRUE
    [7]:
      Name = Warn_ModuleRecovery
      Message = {$AppModule/Recovery.Warning}
      Severity = 0
      Behavior = DiscreteValueMonitoring
        Monitoring:
          MonitoredPV = EM2::RecoveryWarning
          TriggerValues:
            [0] = TRUE
    [8]:
      Name = Alrm_ModuleRecovery
      Message = {$AppModule/Recovery.Alarm}
      Severity = 0
      Behavior = DiscreteValueMonitoring
        Monitoring:
          MonitoredPV = EM2::RecoveryAlarm
          TriggerValues:
            [0] = TRUE
    [9]:
      Name = ModuleInfo
      Message = {$AppModule/Module.Info}
      AdditionalInformation1 = EM2AlarmContent
    [10]:
      Name = ModuleWarning
      Message = {$AppModule/Module.Warning}
      AdditionalInformation1 = EM2AlarmContent
    [11]:
      Name = ModuleAlarm
      Message = {$AppModule/Module.Alarm}
      Code = 1000
      AdditionalInformation1 = EM2AlarmContent
  mapp.AlarmX.Core.Snippets:
    [0]:
      Key = ModuleName
      Value:
        PV = EM2::ModuleName
  mapp.AlarmX.Core.Categories:
    [0]:
      Name = Information
      SourceProperty:
        Severity = 0..99
    [1]:
      Name = Warning
      SourceProperty:
        Severity = 100..199
    [2]:
      Name = Alarm
      SourceProperty:
        Severity = 1000..1199
```

### EM2CFG.mprecipexml - PC/EM2/mappServices/EM2CFG.mprecipexml
```
Element gRecipeXml_EM2 (Type=mprecipexml)
```

### EM2PML.mppackmlmodule - PC/EM2/mappServices/EM2PML.mppackmlmodule
```
Element gPackMLModule_EM2 (Type=mppackmlmodule)
  Module:
    Parent:
      Parent = gMainModule
      Activation = 0
```

### EM3.vvm - PC/EM3/EM3.vvm
```iecst
VAR_CONFIG
	Cyclic#1.::gMainModule AT %Q.EM3::ModuleInterface.MainPml; (*Insert your comment here...*)
	Cyclic#1.EM3::gAlarmXCore_EM3 AT %Q.EM3::ModuleInterface.AlarmCore; (*Insert your comment here...*)
	EM3::gRecipeXml_EM3 AT %Q.EM3::ModuleInterface.RecipeCore; (*Insert your comment here...*)
	EM3::gPackMLModule_EM3 AT %Q.EM3::ModuleInterface.ModulePml; (*Insert your comment here...*)
END_VAR
```

### EM3ALM.mpalarmxcore - PC/EM3/mappServices/EM3ALM.mpalarmxcore
```
Element gAlarmXCore_EM3 (Type=mpalarmxcore)
  mapp.AlarmX.Core:
    Mapping:
      [0]:
        Alarm = Inf*
        [0] = Aggregate
          Name = ModuleInfo
      [1]:
        Alarm = Warn*
        [0] = Aggregate
          Name = ModuleWarning
      [2]:
        Alarm = Alrm*
        [0] = Aggregate
          Name = ModuleAlarm
    Default:
      [0] = Remain
  mapp.AlarmX.Core.Configuration:
    [0]:
      Name = Inf_ModuleOperation
      Message = {$AppModule/Operation.Info}
      Severity = 0
      Behavior = DiscreteValueMonitoring
        Monitoring:
          MonitoredPV = EM3::OperationInformation
          TriggerValues:
            [0] = TRUE
    [1]:
      Name = Warn_ModuleOperation
      Message = {$AppModule/Operation.Warning}
      Severity = 0
      Behavior = DiscreteValueMonitoring
        Monitoring:
          MonitoredPV = EM3::OperationWarning
          TriggerValues:
            [0] = TRUE
    [2]:
      Name = Alrm_ModuleOperation
      Message = {$AppModule/Operation.Alarm}
      Severity = 0
      Behavior = DiscreteValueMonitoring
        Monitoring:
          MonitoredPV = EM3::OperationAlarm
          TriggerValues:
            [0] = TRUE
    [3]:
      Name = Inf_ModuleConfig
      Message = {$AppModule/Configuration.Info}
      Severity = 0
      Behavior = DiscreteValueMonitoring
        Monitoring:
          MonitoredPV = EM3::ConfigInformation
          TriggerValues:
            [0] = TRUE
    [4]:
      Name = Warn_ModuleConfig
      Message = {$AppModule/Configuration.Warning}
      Severity = 0
      Behavior = DiscreteValueMonitoring
        Monitoring:
          MonitoredPV = EM3::ConfigWarning
          TriggerValues:
            [0] = TRUE
    [5]:
      Name = Alrm_ModuleConfig
      Message = {$AppModule/Configuration.Alarm}
      Severity = 0
      Behavior = DiscreteValueMonitoring
        Monitoring:
          MonitoredPV = EM3::ConfigAlarm
          TriggerValues:
            [0] = TRUE
    [6]:
      Name = Inf_ModuleRecovery
      Message = {$AppModule/Recovery.Info}
      Severity = 0
      Behavior = DiscreteValueMonitoring
        Monitoring:
          MonitoredPV = EM3::RecoveryInformation
          TriggerValues:
            [0] = TRUE
    [7]:
      Name = Warn_ModuleRecovery
      Message = {$AppModule/Recovery.Warning}
      Severity = 0
      Behavior = DiscreteValueMonitoring
        Monitoring:
          MonitoredPV = EM3::RecoveryWarning
          TriggerValues:
            [0] = TRUE
    [8]:
      Name = Alrm_ModuleRecovery
      Message = {$AppModule/Recovery.Alarm}
      Severity = 0
      Behavior = DiscreteValueMonitoring
        Monitoring:
          MonitoredPV = EM3::RecoveryAlarm
          TriggerValues:
            [0] = TRUE
    [9]:
      Name = ModuleInfo
      Message = {$AppModule/Module.Info}
      AdditionalInformation1 = EM3AlarmContent
    [10]:
      Name = ModuleWarning
      Message = {$AppModule/Module.Warning}
      AdditionalInformation1 = EM3AlarmContent
    [11]:
      Name = ModuleAlarm
      Message = {$AppModule/Module.Alarm}
      Code = 1000
      AdditionalInformation1 = EM3AlarmContent
  mapp.AlarmX.Core.Snippets:
    [0]:
      Key = ModuleName
      Value:
        PV = EM3::ModuleName
```

### EM3CFG.mprecipexml - PC/EM3/mappServices/EM3CFG.mprecipexml
```
Element gRecipeXml_EM3 (Type=mprecipexml)
```

### EM3PML.mppackmlmodule - PC/EM3/mappServices/EM3PML.mppackmlmodule
```
Element gPackMLModule_EM3 (Type=mppackmlmodule)
  Module:
    Parent:
      Parent = gMainModule
      Activation = 0
```

### EMx.vvm - PC/EMx/EMx.vvm
```iecst
VAR_CONFIG
	Cyclic#1.::gMainModule AT %Q.EMx::ModuleInterface.MainPml; (*Insert your comment here...*)
	EMx::gAlarmXCore_EMx AT %Q.EMx::ModuleInterface.AlarmCore; (*Insert your comment here...*)
	EMx::gPackMLModule_EMx AT %Q.EMx::ModuleInterface.ModulePml; (*Insert your comment here...*)
	EMx::gRecipeXml_EMx AT %Q.EMx::ModuleInterface.RecipeCore; (*Insert your comment here...*)
END_VAR
```

### EMxALM.mpalarmxcore - PC/EMx/mappServices/EMxALM.mpalarmxcore
```
Element gAlarmXCore_EMx (Type=mpalarmxcore)
  mapp.AlarmX.Core:
    Mapping:
      [0]:
        Alarm = Inf*
        [0] = Aggregate
          Name = ModuleInfo
      [1]:
        Alarm = Warn*
        [0] = Aggregate
          Name = ModuleWarning
        [1]
      [2]:
        Alarm = Alrm*
        [0] = Aggregate
          Name = ModuleAlarm
    Default:
      [0] = Remain
  mapp.AlarmX.Core.Configuration:
    [0]:
      Name = Inf_ModuleProcess
      Message = {$AppModuleEMx/Process.Info}
      Severity = 0
      Behavior = DiscreteValueMonitoring
        Monitoring:
          MonitoredPV = EMx::ProcessInformation
          TriggerValues:
            [0] = TRUE
    [1]:
      Name = Warn_ModuleProcess
      Message = {$AppModuleEMx/Process.Warning}
      Severity = 0
      Behavior = DiscreteValueMonitoring
        Monitoring:
          MonitoredPV = EMx::ProcessWarning
          TriggerValues:
            [0] = TRUE
    [2]:
      Name = Alrm_ModuleProcess
      Message = {$AppModuleEMx/Process.Alarm}
      Severity = 0
      Behavior = DiscreteValueMonitoring
        Monitoring:
          MonitoredPV = EMx::ProcessAlarm
          TriggerValues:
            [0] = TRUE
    [3]:
      Name = ModuleInfo
      Message = {$AppModuleEMx/Module.Info}
      AdditionalInformation1 = EMxAlarmContent
    [4]:
      Name = ModuleWarning
      Message = {$AppModuleEMx/Module.Warning}
      Code = 100
      AdditionalInformation1 = EMxAlarmContent
    [5]:
      Name = ModuleAlarm
      Message = {$AppModule/Module.Alarm}
      Code = 1000
      AdditionalInformation1 = EMxAlarmContent
  mapp.AlarmX.Core.Snippets:
    [0]:
      Key = ModuleName
      Value:
        PV = EMx::ModuleName
  mapp.AlarmX.Core.Categories:
    [0]:
      Name = Information
      SourceProperty:
        Severity = 0..99
    [1]:
      Name = Warning
      SourceProperty:
        Severity = 100..199
    [2]:
      Name = Alarm
      SourceProperty:
        Severity = 1000..1199
```

### EMxCFG.mprecipexml - PC/EMx/mappServices/EMxCFG.mprecipexml
```
Element gRecipeXml_EMx (Type=mprecipexml)
```

### EMxPML.mppackmlmodule - PC/EMx/mappServices/EMxPML.mppackmlmodule
```
Element gPackMLModule_EMx (Type=mppackmlmodule)
  Module:
    Parent:
      Parent = gMainModule
      Activation = 0
```

### EM2.vvm - PC/ReusedModules/EM2/EM2.vvm
```iecst
VAR_CONFIG
	Cyclic#1.::gMainModule AT %Q.EM2::ModuleInterface.MainPml; (*Insert your comment here...*)
END_VAR
```

### EM3.vvm - PC/ReusedModules/EM3/EM3.vvm
```iecst
VAR_CONFIG
	Cyclic#1.::gMainModule AT %Q.EM3::ModuleInterface.MainPml; (*Insert your comment here...*)
END_VAR
```

### TrackMod.vvm - PC/TrackMod/TrackMod.vvm
```iecst
VAR_CONFIG
	Cyclic#1.::gSampleTrak_SectorTrackA AT %Q.TrackMod::TrackInterface.SectorTrackA; (*Insert your comment here...*)
	Cyclic#1.::gSampleTrak AT %Q.TrackMod::TrackInterface.SampleTrak; (*Insert your comment here...*)
	Cyclic#1.TrackMod::gTrackModule AT %Q.TrackMod::TrackInterface.ModulePml; (*Insert your comment here...*)
	Cyclic#1.TrackMod::gAlarmXCore_TrackModule AT %Q.TrackMod::TrackInterface.AlarmCore; (*Insert your comment here...*)
	Cyclic#1.TrackMod::gRecipeXml_TrackModule AT %Q.TrackMod::TrackInterface.RecipeCore; (*Insert your comment here...*)
END_VAR
```

### TrakALM.mpalarmxcore - PC/TrackMod/mappServices/TrakALM.mpalarmxcore
```
Element gAlarmXCore_TrackModule (Type=mpalarmxcore)
  mapp.AlarmX.Core:
    Mapping:
      [0]:
        Alarm = Inf*
        [0] = Aggregate
          Name = TrakModuleInfo
      [1]:
        Alarm = Warn*
        [0] = Aggregate
          Name = TrakModuleWarning
      [2]:
        Alarm = Alrm*
        [0] = Aggregate
          Name = TrakModuleAlarm
    Default:
      [0] = Remain
      [1] = Reaction
        Name = TrakTest
  mapp.AlarmX.Core.Configuration:
    [0]:
      Name = Alrm_ErrorStop
      Message = {$TrakAssembly/TrakErrorStop}
      Code = 1000
      Behavior = DiscreteValueMonitoring
        Monitoring:
          MonitoredPV = TrackMod::AsmSampleT:fbAsmReadStatus.AssemblyErrorStop
          TriggerValues:
            [0] = TRUE
    [1]:
      Name = Inf_PowerOn
      Message = {$TrakAssembly/TrakPowerOn}
      Behavior = DiscreteValueMonitoring
        Monitoring:
          MonitoredPV = TrackMod::AsmSampleT:fbAsmReadInfo.AssemblyInfo.PowerOn
          TriggerValues:
            [0] = TRUE
    [2]:
      Name = Inf_ModuleTest
      Message = {$TrakAssembly/LocalTrakModuleInfo}
      Severity = 0
      Behavior = DiscreteValueMonitoring
        Monitoring:
          MonitoredPV = TrackMod::AsmAlarm:TriggerTestInformation
          TriggerValues:
            [0] = TRUE
    [3]:
      Name = Warn_ModuleTest
      Message = {$TrakAssembly/LocalTrakModuleWarning}
      Code = 100
      Severity = 50
      Behavior = DiscreteValueMonitoring
        Monitoring:
          MonitoredPV = TrackMod::AsmAlarm:TriggerTestWarning
          TriggerValues:
            [0] = TRUE
    [4]:
      Name = Alrm_ModuleTest
      Message = {$TrakAssembly/LocalTrakModuleAlarm}
      Code = 1000
      Severity = 100
      Behavior = DiscreteValueMonitoring
        Monitoring:
          MonitoredPV = TrackMod::AsmAlarm:TriggerTestAlarm
          TriggerValues:
            [0] = TRUE
    [5]:
      Name = TrakModuleInfo
      Message = {$TrakAssembly/Module.Info}
      AdditionalInformation1 = trackAlarmContent
    [6]:
      Name = TrakModuleWarning
      Message = {$TrakAssembly/Module.Warning}
      Code = 100
      AdditionalInformation1 = trackAlarmContent
    [7]:
      Name = TrakModuleAlarm
      Message = {$TrakAssembly/Module.Alarm}
      Code = 1000
      AdditionalInformation1 = trackAlarmContent
  mapp.AlarmX.Core.Snippets:
    [0]:
      Key = ModuleName
      Value:
        PV = TrackMod::ModuleName
  mapp.AlarmX.Core.Categories:
    [0]:
      Name = Information
      SourceProperty:
        Severity = 0..99
    [1]:
      Name = Warning
      SourceProperty:
        Severity = 100..199
    [2]:
      Name = Alarm
      SourceProperty:
        Severity = 1000..1199
```

### TrakCFG.mprecipexml - PC/TrackMod/mappServices/TrakCFG.mprecipexml
```
Element gRecipeXml_TrackModule (Type=mprecipexml)
  Alarms = MpAlarmX
Element gMpRecipeDiagXml (Type=mprecipexml)
```

### TrakPML.mppackmlmodule - PC/TrackMod/mappServices/TrakPML.mppackmlmodule
```
Element gTrackModule (Type=mppackmlmodule)
  Module:
    Name = TrackAssembly
    Parent:
      Parent = gMainModule
      Activation = 0
```
